		(*Echo OFF*)
		sEchoOff:='ATE0';
		sEchoOff:=CONCAT(sEchoOff,'X');	(*The "X" is a placeholder in the send-string
										for the "CR" (Hex 0D) in the send-Array*)
		MEMCPY(ADR(arEchoOff),ADR(sEchoOff),LEN(sEchoOff)); (*Copy String to ARRAY*)
		arEchoOff[LEN(sEchoOff)]:=16#0D;(*Place the "CR" in the array*)

		(*Mode Text*)
		sLogin:='AT+CMGF=';
		sLogin:=CONCAT(sLogin,'1');
		sLogin:=CONCAT(sLogin,'X');	(*The "X" is a placeholder in the send-string
										for the "CR" (Hex 0D) in the send-Array*)
		MEMCPY(ADR(arLogin),ADR(sLogin),LEN(sLogin)); (*Copy String to ARRAY*)
		arLogin[LEN(sLogin)]:=16#0D;	(*Place the "CR" in the array*)

		nStep	:= 100;


	100:(*Turn Off the Echo*)
		fbSendData(
		pSendData:=ADR(arEchoOff),
		Length:= LEN(sEchoOff),
		TXbuffer:= stTxBuffer);

		IF NOT fbSendData.Busy THEN
			nStep:=110;
		END_IF

		IF  fbSendData.Error<>0 THEN
			bError:= TRUE;
			nErrorID:= fbSendData.Error;
			nStep:=1000;
		END_IF


	110:(*Wait explicitly (by Prefix) for an "OK"-Answer,
		because the echo may still be on or is already switched off, so the answer may differ in length.
		Only ok is possible, any other answer caused by Comm-Error will end in global timeout*)

		fbReceiveData(
		pPrefix:= ADR(arAnswerOK),
		LenPrefix:= 2,
		pReceiveData:= ADR(arEchoOffAnswerRcv),
		SizeReceiveData:= SIZEOF(arEchoOffAnswerRcv),
		Timeout:= t#500ms,
		RXbuffer:= stRxBuffer);

		(*Telegram is received*)
		IF 			fbReceiveData.DataReceived
			AND NOT fbReceiveData.busy
			AND		(arEchoOffAnswerRcv[1]=arAnswerOK[1])
			AND 	(arEchoOffAnswerRcv[2]=arAnswerOK[2])	THEN
						nStep:=200;
		END_IF


	200:(*Send AT+CMGF Command*)
		fbSendData(
		pSendData:=ADR(arLogin),
		Length:= LEN(sLogin),
		TXbuffer:= stTxBuffer);

		IF NOT fbSendData.Busy THEN
			nStep:=210;
		END_IF

		IF  fbSendData.Error<>0 THEN
			bError:= TRUE;
			nErrorID:= fbSendData.Error;
			nStep:=1000;
		END_IF


	210:(*Wait for OK or Err-Answer. Any other answer caused by Comm-Error will end in global timeout*)
		(*Do NOT remove the "0" prefix, because the FB is used previously*)
		fbReceiveData(
		pPrefix:= 0,
		LenPrefix:= 0,
		pReceiveData:= ADR(arLoginAnswerRcv),
		SizeReceiveData:= SIZEOF(arLoginAnswerRcv),
		Timeout:= t#500ms,
		RXbuffer:= stRxBuffer);

		(*Telegram is received*)
		IF 	(fbReceiveData.DataReceived	AND NOT 	fbReceiveData.busy)	THEN
				nStep:=220;
		END_IF


	220:(*Analyze answer*)
		IF		(arLoginAnswerRcv[3]=arAnswerOK[1]) AND (arLoginAnswerRcv[4]=arAnswerOK[2])	THEN
					nStep:=1000;		(*Login successful*)
		ELSIF	(arLoginAnswerRcv[3]=arAnswerErr[1]) AND (arLoginAnswerRcv[4]=arAnswerErr[2])	THEN
					bError:= TRUE;
					nErrorID:= 16#8004;	(*Login failed due to wrong PIN or no Card or already logged in*)
					nStep:=1000;
		ELSE
					bError:= TRUE;
					nErrorID:= 16#8005;	(*Undefined answer*)
					nStep:=1000;
		END_IF


	900:(*Timeout*)
		bError:= TRUE;
		nErrorID:= 16#8001;
		nStep:=1000;


	1000:(*Reset Receive-FB*)
		fbReceiveData(	Reset:=TRUE,RXbuffer:= stRxBuffer);
		tonWaitTime(IN:=TRUE, PT:=t#1000ms);
		IF	tonWaitTime.Q	THEN
			tonWaitTime(IN:=FALSE);
			fbReceiveData(	Reset:=FALSE,RXbuffer:= stRxBuffer);
			nStep:=1010;
		END_IF


	1010:(*Send/Receive successful -> Reset FBs*)
		fbClearComBuffer(buffer:=stRxBuffer);
		fbClearComBuffer(buffer:=stTxBuffer);
		tonWaitTime(IN:=TRUE, PT:=t#1000ms);
		IF	tonWaitTime.Q	THEN
			tonWaitTime(IN:=FALSE);
			nStep:=0;
			bBusy:=FALSE;
		END_IF

	END_CASE;

END_FUNCTION_BLOCK

// ---- 00_FunctionsBlocks/Common/DataProcessing/FB_XorWord.TcPOU
FUNCTION_BLOCK FB_XorWord
// Takes in a Word and its past value and input the bits that have changed and the bits active in 2 arrays of array of bool
VAR_INPUT
	MyNewWord	:WORD;      //Mon nouveau AlarmCode actualisée a chaque temps de Cycle
	MyWord		:WORD;		// AlarmCode du cycle précedent
END_VAR
VAR_OUTPUT
	XORarray 	:ARRAY [0..15] OF BOOL;  //Tableau avec les bits qui ont subit une modif entre MyNewWord et MyWord
	Boolarray	:ARRAY [0..15] OF BOOL; // MyNewWord convertis en Array of BOOL
END_VAR
VAR
	MyXorWord:WORD;
	FB_Word_TO_Bool : FB_WordToArrayOfBool;
END_VAR

// Operateur XOR pour trouver les Bits modifiés
MyXorWord:= Myword XOR MyNewWord;

FB_Word_TO_Bool(MyWord:=MyXorWord,ArrayOfBool=>XORarray);
FB_Word_TO_Bool(MyWord:=MyNewWord,ArrayOfBool=>Boolarray);

END_FUNCTION_BLOCK

// ---- 00_FunctionsBlocks/Common/BoolManagement/FB_WordToArrayOfBool.TcPOU
FUNCTION_BLOCK FB_WordToArrayOfBool
// Transforms a Word in an array of BOOL;
VAR_INPUT
	MyWord	:WORD;
END_VAR
VAR_OUTPUT
	ArrayOfBool: ARRAY [0..15] OF BOOL;
END_VAR

ArrayOfBool[0] := BIT_TO_BOOL(MyWord.0);
ArrayOfBool[1] := BIT_TO_BOOL(MyWord.1);
ArrayOfBool[2] := BIT_TO_BOOL(MyWord.2);
ArrayOfBool[3] := BIT_TO_BOOL(MyWord.3);
ArrayOfBool[4] := BIT_TO_BOOL(MyWord.4);
ArrayOfBool[5] := BIT_TO_BOOL(MyWord.5);
ArrayOfBool[6] := BIT_TO_BOOL(MyWord.6);
ArrayOfBool[7] := BIT_TO_BOOL(MyWord.7);
ArrayOfBool[8] := BIT_TO_BOOL(MyWord.8);
ArrayOfBool[9] := BIT_TO_BOOL(MyWord.9);
ArrayOfBool[10] := BIT_TO_BOOL(MyWord.10);
ArrayOfBool[11] := BIT_TO_BOOL(MyWord.11);
ArrayOfBool[12] := BIT_TO_BOOL(MyWord.12);
ArrayOfBool[13] := BIT_TO_BOOL(MyWord.13);
ArrayOfBool[14] := BIT_TO_BOOL(MyWord.14);
ArrayOfBool[15] := BIT_TO_BOOL(MyWord.15);

END_FUNCTION_BLOCK

// ---- 00_FunctionsBlocks/Beckhoff/Communication/SMS/FB_Extract_Num_Mes.TcPOU
FUNCTION_BLOCK FB_Extract_Num_Mes
// extract phone number from the received message
VAR_INPUT
    InMessage     : STRING(255);
END_VAR
VAR_OUTPUT
    OutDataEntry  :ST_SMSDataSetEntry_Read;
END_VAR
VAR
    ChaineTmp     : STRING(255);
    Num           : STRING(255);
    Pos           : INT;
    Pos1          : INT;
    Pos2          : INT;
    Pos3          : INT;    
	Offset		: INT ; 
END_VAR

//+CMGR: "REC UNREAD","+33776039883",,"18/04/19,18:25:44+08"$R$NBonjour je m'appelle henry$R$N 50
Pos:=FIND(InMessage,',"');
chaineTmp:=MID(InMessage,LEN(InMessage)-21,POS+2);
Pos1:=FIND(chaineTmp,'",,');
Num:=MID(chaineTmp,Pos1-1,1);
Pos3:= FIND(Num,'+');
OutDataEntry.Num:= SEL(Pos3= 0 ,Num ,CONCAT(STR1:= CstPhoneIndicator_G, STR2:= Num) );
Pos2:=FIND(InMessage,'$R$N');
Offset := FIND(MID(InMessage,LEN(InMessage)-Pos2,Pos2+2),'$R$N') ;


OutDataEntry.Message:=MID(InMessage,Offset-1,Pos2+2);//OutDataEntry.Message:=MID(InMessage,LEN(InMessage)-Pos2-3,LEN(InMessage));	// OutDataEntry.Message:=MID(InMessage,LEN(InMessage)-Pos2-3,Pso2+2);

END_FUNCTION_BLOCK

// ---- 04_Application/MAIN/TEST.TcPOU
PROGRAM TEST
VAR
// create an instance for all FB in base project in order to test if there are errors in the FB ()

	moyenne_test : MOYENNE;
	time_Test : TIME := T#5s;
	bTest : BOOL;
	rValue : REAL;

(*
FB_PM_PM5XXX						: FB_PM_PM5XXX ; 
FB_GRID_PLAN						: FB_GRID_PLAN ; 	
FB_CB_AuxMVCB						:FB_CB_AuxMVCB						;
FB_CB_FeederMVCB            		:FB_CB_FeederMVCB            		 ;
FB_CB_GridMVCB               		:FB_CB_GridMVCB               		;
FB_CB_MainHVCB           			:FB_CB_MainHVCB           			;
FB_CB_MainMVCB           			:FB_CB_MainMVCB           			;
FB_CB_MeasureMVCB        			:FB_CB_MeasureMVCB        			;
FB_CB_MVSwitch           	  		:FB_CB_MVSwitch;             		
FB_CB_Switch	               		:FB_CB_Switch;               		
FB_Fan_Basic                		:FB_Fan_Basic                		 ;
FB_FSS                      		:FB_FSS                      		 ;
FB_GRID_Enedis              		:FB_GRID_Enedis              		 ;
FB_GRID_MADI                		:FB_GRID_MADI                		 ;
FB_HVAC_Standard            		:FB_HVAC_Standard            		          ;
FB_HVAC_MADI                		:FB_HVAC_MADI                		 ;
FB_PM_520x230               		:FB_PM_520x230               		 ;
FB_PM_A40                   		:FB_PM_A40                   		 ;
FB_PM_ION7650               		:FB_PM_ION7650               		 ;
FB_PM_Janitza               		:FB_PM_Janitza               		 ;
FB_PM_PM3250                		:FB_PM_PM3250                		 ;
FB_PM_SM103E                		:FB_PM_SM103E                		 ;
FB_ProtectRelay_DM2     			:FB_ProtectRelay_DM2     		;
FB_ProtectRelay_PACE100ST    		:FB_ProtectRelay_PACE100ST    		;
FB_ProtectRelay_REF615       		:FB_ProtectRelay_REF615       		;
FB_ProtectRelay_SEPAM10a     		:FB_ProtectRelay_SEPAM10a     		;
FB_ProtectRelay_SepamS48     		:FB_ProtectRelay_SepamS48     		;
FB_ProtectRelay_SepamT20     		:FB_ProtectRelay_SepamT20     		;
FB_ProtectRelay_VIP410       		:FB_ProtectRelay_VIP410       		;
FB_ProtectRelay_WIP1         		:FB_ProtectRelay_WIP1         		;
FB_ANA_Irra_Fx               		:FB_ANA_Irra_Fx               		;
FB_ANA_SMP1X                 		:FB_ANA_SMP1X                 		;
FB_ANA_AllInOne              		:FB_ANA_AllInOne              		    ;
FB_TOR_CB                    		:FB_TOR_CB                    		;
FB_TOR_DS                    		:FB_TOR_DS                    		;
FB_TOR_ES                    		:FB_TOR_ES                    		;
FB_TOR_Fuse                  		:FB_TOR_Fuse                  		;
FB_TOR_Rain                			:FB_TOR_Rain                			;
FB_TOR_SD                    		:FB_TOR_SD                    		;
FB_TOR_Spd                   		:FB_TOR_Spd                   		;
FB_TOR_ToS                   		:FB_TOR_ToS                   		;
FB_EM_Pulse                  		:FB_EM_Pulse                  		      ;
FB_Transfo_HVCom             		:FB_Transfo_HVCom             		;
FB_Transfo_MV                		:FB_Transfo_MV                		;
FB_Transfo_MVCom             		:FB_Transfo_MVCom             		;
FB_UPS_CXC                   		:FB_UPS_CXC                   		;
FB_UPS_ENERIS                		:FB_UPS_ENERIS                		;
FB_BAT_KP_MK1						: FB_BAT_KP_MK1					; 
//FB_BAT_M3							: FB_BAT_M3       					;          
FB_BAT_Saft                 		: FB_BAT_Saft                      ;
FB_BAT_Sams                 		: FB_BAT_Sams                      ;

FB_Datalogger_SchSkid       		: FB_Datalogger_SchSkid            ;

FB_HVAC_MeAcMbs1            		: FB_HVAC_MeAcMbs1                 ;
*)
FB_INV_Huawei_SL            		: FB_INV_Huawei_SL                 ;

FB_INV_Huawei_Sun2000KtlMo  		: FB_INV_Huawei_Sun2000KtlMo       ;
FB_INV_JemaIFX6             		: FB_INV_JemaIFX6                  ;
FB_INV_Power_One            		: FB_INV_Power_One                 ;
FB_INV_Sch4400              		: FB_INV_Sch4400                   ;
FB_INV_SmaSCXXXXCP_HE       		: FB_INV_SmaSCXXXXCP_HE            ;
FB_INV_SmaSCXXXXUP_US       		: FB_INV_SmaSCXXXXUP_US            ;
(*
FB_IPC                      		: FB_IPC                           ;
FB_PM_Digiware              		: FB_PM_Digiware                   ;
FB_PM_PM800                 		: FB_PM_PM800                      ;
FB_PM_Prometer              		: FB_PM_Prometer                   ;
FB_PM_Q100                  		: FB_PM_Q100                       ;
FB_PCS_Jema_IBX3            		: FB_PCS_Jema_IBX3                 ;
FB_PCS_PE                   		: FB_PCS_PE                        ;
FB_PCS_Sma_SCS3450UP        		: FB_PCS_Sma_SCS3450UP             ;
FB_PPC_SmaKita              		: FB_PPC_SmaKita                   ;
FB_ProtectRelay_Siprotec    	    : FB_ProtectRelay_Siprotec         ;
FB_ProtectRelay_Flair23DM   	    : FB_ProtectRelay_Flair23DM        ;
FB_ProtectRelay_MaxI        	    : FB_ProtectRelay_MaxI             ;
FB_ProtectRelay_NSXCB       	    : FB_ProtectRelay_NSXCB            ;
FB_Router                   	    : FB_Router                        ;
FB_ANA_IO                   	    : FB_ANA_IO                        ;
FB_ANA_DustIQ               	    : FB_ANA_DustIQ                    ;

FB_TOR_Digicode             	    : FB_TOR_Digicode                  ;
FB_TOR_Standard             	    : FB_TOR_Standard                  ;
FB_TOR_MS                   	    : FB_TOR_MS                        ;
FB_TOR_VP                   	    : FB_TOR_VP                        ;
FB_TAC                      	    : FB_TAC                           ;
FB_NCU_Axial                	    : FB_NCU_Axial                     ;
FB_UPS_PS10048              	    : FB_UPS_PS10048                   ;
FB_PM_ION9200						: FB_PM_ION9200 ; 	
	

FB_PPC_PE							: FB_PPC_PE ; 
FB_UPS_MCSU4 						: FB_UPS_MCSU4 ; 
FB_ProtectRelay_SMNS7SL86 			: FB_ProtectRelay_SMNS7SL86 ; 
*)
FB_INV_PE_HEMK : FB_INV_PE_HEMK ; 
	FB_INV_PE_HEMG3 : FB_INV_PE_HEMG3 ; 
END_VAR


moyenne_test(
	In_fenetre_mesure := time_Test,
	In_synchro := CalLocalTimeStruct.wSecond MOD 5 = 0,
	In_valeur := word_to_real(CalLocalTimeStruct.wSecond)
);
moyenne_test.Calcul();

(*
FB_GRID_PLAN.M_Execute() ; 
FB_CB_AuxMVCB.M_Execute() ; 					
FB_CB_FeederMVCB.M_Execute() ; 			            	
FB_CB_GridMVCB.M_Execute() ; 			               	
FB_CB_MainHVCB.M_Execute() ; 			           		
FB_CB_MainMVCB.M_Execute() ; 			           		
FB_CB_MeasureMVCB.M_Execute() ; 			        		
FB_CB_MVSwitch.M_Execute() ; 			             	
FB_CB_Switch.M_Execute() ; 			               	
FB_Fan_Basic.M_Execute() ; 		                	
FB_FSS.M_Execute() ; 		                      	
FB_GRID_Enedis.M_Execute() ; 		              	
FB_GRID_MADI.M_Execute() ; 		                	
FB_HVAC_Standard.M_Execute() ; 		            	
FB_HVAC_MADI.M_Execute() ; 		                	
FB_PM_520x230.M_Execute() ; 		               	
FB_PM_A40.M_Execute() ; 		                   	
FB_PM_ION7650.M_Execute() ; 		               	
FB_PM_Janitza.M_Execute() ; 		               	
FB_PM_PM3250.M_Execute() ; 		                	
FB_PM_SM103E.M_Execute() ; 		                	
FB_ProtectRelay_DM2.M_Execute() ; 		     		
FB_ProtectRelay_PACE100ST.M_Execute() ; 		    	
FB_ProtectRelay_REF615.M_Execute() ; 		       	
FB_ProtectRelay_SEPAM10a.M_Execute() ; 		     	
FB_ProtectRelay_SepamS48.M_Execute() ; 		     	
FB_ProtectRelay_SepamT20.M_Execute() ; 		     	
FB_ProtectRelay_VIP410.M_Execute() ; 		       	
FB_ProtectRelay_WIP1.M_Execute() ; 		         	
FB_ANA_Irra_Fx.M_Execute() ; 		               	
FB_ANA_SMP1X.M_Execute() ; 		                 	
FB_ANA_AllInOne.M_Execute() ; 		              	
FB_TOR_CB.M_Execute() ; 		                    	
FB_TOR_DS.M_Execute() ; 		                    	
FB_TOR_ES.M_Execute() ; 		                    	
FB_TOR_Fuse.M_Execute() ; 		                  	
FB_TOR_Rain.M_Execute() ; 		                		
FB_TOR_SD.M_Execute() ; 		                    	
FB_TOR_Spd.M_Execute() ; 		                   	
FB_TOR_ToS.M_Execute() ; 		                   	
FB_EM_Pulse.M_Execute() ; 		                  	
FB_Transfo_HVCom.M_Execute() ; 		             	
FB_Transfo_MV.M_Execute() ; 		                	
FB_Transfo_MVCom.M_Execute() ; 		             	
FB_UPS_CXC.M_Execute() ; 		                   	
FB_UPS_ENERIS.M_Execute() ; 		                	
FB_BAT_KP_MK1.M_Execute() ; 							
FB_BAT_M3.M_Execute() ; 								
FB_BAT_Saft.M_Execute() ; 		                 	
FB_BAT_Sams.M_Execute() ; 		                 	
FB_Datalogger_IOWIT.M_Execute() ; 		         	
FB_Datalogger_PPCVerrerie.M_Execute() ; 		   	
FB_Datalogger_SchSkid.M_Execute() ; 		       	
FB_Datalogger_SENECA.M_Execute() ; 		        	
FB_HVAC_MeAcMbs1.M_Execute() ; 		            	
*)
FB_INV_Huawei_SL.M_Execute() ; 		            	
FB_INV_Huawei_Sun2000KtlMo.M_Execute() ; 		  	
FB_INV_JemaIFX6.M_Execute() ; 		             	
FB_INV_Power_One.M_Execute() ; 		            	
FB_INV_Sch4400.M_Execute() ; 		              	
FB_INV_SmaSCXXXXCP_HE.M_Execute() ; 		       	
FB_INV_SmaSCXXXXUP_US.M_Execute() ; 		       	


(*
FB_IPC.M_Execute() ; 		                      	
FB_PM_Digiware.M_Execute() ; 		              	
FB_PM_PM800.M_Execute() ; 		                 	
FB_PM_Prometer.M_Execute() ; 		              	
FB_PM_Q100.M_Execute() ; 		                  	
FB_PCS_Jema.M_Execute() ; 		                 	
FB_PCS_Jema_IBX3.M_Execute() ; 		            	
FB_PCS_PE.M_Execute() ; 		                   	
FB_PCS_Sma_SCS3450UP.M_Execute() ; 		       	
FB_PPC_SmaKita.M_Execute() ; 		              	
FB_ProtectRelay_Siprotec.M_Execute() ; 		    	
FB_ProtectRelay_Flair23DM.M_Execute() ; 		   	
FB_ProtectRelay_MaxI.M_Execute() ; 		        	
FB_ProtectRelay_NSXCB.M_Execute() ; 		       	
FB_Router.M_Execute() ; 		                   	
FB_ANA_IO.M_Execute() ; 		                   	
FB_ANA_Irra_Fx.M_Execute() ; 		              	
FB_ANA_DustIQ.M_Execute() ; 		               	
FB_ANA_SMP1X.M_Execute() ; 		               	
FB_TOR_Digicode.M_Execute() ; 		             	
FB_TOR_Standard.M_Execute() ; 		             	
FB_TOR_MS.M_Execute() ; 		                   	
FB_TOR_VP.M_Execute() ; 		                   	
FB_TAC.M_Execute() ; 		                      	
FB_EM_Pulse.M_Execute() ; 		                 	
FB_NCU_Axial.M_Execute() ; 		                	
FB_UPS_PS10048.M_Execute() ; 		              	
FB_PM_PM5XXX.M_Execute() ; 
FB_PM_ION9200.M_Execute() ; 
FB_PPC_PE.M_Execute() ; 

				  				
FB_UPS_MCSU4.M_Execute() ;  				
FB_ProtectRelay_SMNS7SL86.M_Execute() ;  	
*)
FB_INV_PE_HEMG3.M_Execute() ;  
FB_INV_PE_HEMK.M_Execute();

END_PROGRAM

// ---- 00_FunctionsBlocks/Beckhoff/DataProcessing/MOYENNE.TcPOU
FUNCTION_BLOCK MOYENNE
VAR_INPUT
	In_valeur: REAL;
	In_synchro: BOOL;
	In_fenetre_mesure: TIME;
END_VAR
VAR_OUTPUT
	Out_fenetre_mesure: TIME;
	Out_fin: BOOL;
	Out_Moyenne_0: REAL;
	Out_Moyenne_1: REAL;
END_VAR
VAR
	F_Fenetre_mesure_active: F_TRIG;
	R_In_Synchro: R_TRIG;
	TOF_0: TOF;
	Fenetre_mesure_active: BOOL;
	Nbr_valeur_mesure: REAL;
END_VAR

ACTION Calcul:
(* Gestion des fronts montants et front descendants *)

	R_In_Synchro(CLK := In_Synchro);
	F_Fenetre_mesure_active(CLK := Fenetre_mesure_active);

(* Traitements *)

	IF R_In_Synchro.Q THEN  (* Initialisation des valeurs au lancement de la synchronisation *)
	
		Out_fin:=False; 
		Nbr_valeur_mesure:=0.0; (* RAZ nbr de cycle automate *)
	
	END_IF;
	

	TOF_0 (IN := R_In_Synchro.Q,(* Gestion de la fenêtre de mesure  *)
		  PT := In_fenetre_mesure,
		  Q => Fenetre_mesure_active,
		  ET => Out_fenetre_mesure);
	
	IF Fenetre_mesure_active  THEN (* Traitement durant la fenêtre de mesure *) 
		
		Out_Moyenne_0:=(Out_Moyenne_0*Nbr_valeur_mesure+In_valeur)/(Nbr_valeur_mesure+1.0); (* calcul moyenne *)
	
		Nbr_valeur_mesure:=Nbr_valeur_mesure+1.0; (* calcul nbr de cycle automate *)
	
	ELSIF F_Fenetre_mesure_active.Q THEN (* Traitement en fin de fenêtre de mesure *)
	
		Out_fin:=true;
		Out_Moyenne_1:=Out_Moyenne_0; (* Sauvegarde de la moyenne calculée *)
		Out_Moyenne_0:=0.0; (* RAZ moyenne calculée *)
	
	End_if;
END_ACTION

END_FUNCTION_BLOCK

// ---- 01_Equipement_Library/Inverter/FB_INV_Huawei_SL.TcPOU
FUNCTION_BLOCK FB_INV_Huawei_SL EXTENDS FB_INV_Base
//////////////////
// SmartLogger Huawei
//////////////////

VAR_INPUT PERSISTENT
	// Parameters of the Object (instance specific)
	{attribute 'OPC.UA.DA' := '1'}  
	ParamIpAddress		   : STRING 	:= '127.0.0.1'; (* (NA)Config: IP Adress of PV INverter*)
	{attribute 'OPC.UA.DA' := '1'} 
	ParamUnitID 			: BYTE  := 0; 			  	(* (NA)   Modbus Unit ID. *)
	ParamNbINV				: BYTE:=1 ; 				(* Number of inverters behind the smartlogger *)
	{attribute 'OPC.UA.DA' := '1'}              		
	ParamnTcpPort			: UINT := 502;				(* TCP port number *)
	ParamPnomINV			: REAL:=60; 				(* (kW) Nominal Power For one inverter *)
	ParamSLNum				: BYTE ; 					(* (NA) Config :Numerous of the ESS in the PP*)
	ParamID_PTR				: UINT;						(* (NA) ID of the PTR where Smartlogger is located*)
	
	
		MesDataExd	AT %Q*		: INV_Huawei_SL;
	
END_VAR

VAR_OUTPUT
	//Child objects
	
END_VAR

VAR

	// M_READ VARIABLES//


//		FB_ModbusRead_I1          	: ARRAY[1..CstNbINVperPTR_G] OF  FB_ModbusRead ; 		// (NA) FB for Modbus Reading
		FB_ModbusRead_I2          	: FB_ModbusRead ; 										// (NA) FB for Modbus Reading
		FB_ModbusRead_I3          	: FB_ModbusRead ; 										// (NA) FB for Modbus Reading
			
//		MesBlock1_Temp 				: ARRAY[1..CstNbINVperPTR_G] OF ARRAY[0..24]  OF WORD; 	// (NA) Temporary Block with multiple modbus reading (Caution : Double Word variables)
//		MesBlock1_Temp 				: ARRAY[0..25*CstNbINVperPTR_G-1]  OF WORD; 			// (NA) Temporary Block with multiple modbus reading (Caution : Double Word variables)
		MesBlock2_Temp 				: ARRAY[0..56] OF WORD;									// (NA) Temporary Block with multiple modbus reading (Caution : Double Word variables)
		MesBlock3_Temp 				: ARRAY[0..14] OF WORD;									// (NA) Temporary Block with multiple modbus reading (Caution : Double Word variables)
                                                                                    		
		                                                                            		
//		MesModbusReadAlarm 		  	: ARRAY[1..CstNbINVperPTR_G] OF BOOL ; 					// (NA) Modbus Read Alarm for all modbus frames		
		MesModbusReadAlarm2 		: BOOL ; 												// (NA) Modbus Read Alarm for all modbus frames			
		MesModbusReadAlarm3 		: BOOL ; 												// (NA) Modbus Read Alarm for all modbus frames			

//		MesModbusAlarmCode			: ARRAY[1..CstNbINVperPTR_G] OF UDINT;					// (NA) Modbus Read Alarm Code
		MesModbusAlarmCode2			: UDINT;												// (NA) Modbus Read Alarm Code
		MesModbusAlarmCode3			: UDINT;												// (NA) Modbus Read Alarm Code

	
	// M_CURTAIL VARIABLES //
		FB_ModbusWrite_I2 		  	: FB_ModbusWrite ; 										// (NA) Functionnal Block for Writing Curtail limit through modbus
		FB_ModbusWrite_I3 		  	: FB_ModbusWrite ; 										// (NA) Functionnal Block for Writing Curtail limit through modbus	
		MesModbusWriteCode          : UDINT ; 												// (NA) Modbus Write Alarm Code 			 
		MesModbusWriteCode2         : UDINT ; 												// (NA) Modbus Write Alarm Code 
	                                                                           		
		MesModbusCurtailAlarm		: BOOL ;				   								// (NA) Modbus Write Curtail Alarm 
		MesModbusCurtailAlarm2		: BOOL ;				   								// (NA) Modbus Write Curtail Alarm 
		WriteBlock_Temp 	AT %Q*	: ARRAY[0..3] OF WORD;				 					// Temporary Block with multiple modbus writing	 
		
END_VAR

METHOD M_AlarmManagement
//////////////////
// Manages IntelliGen Alarms
/////////////////

VAR 
	// Method local variables (reinitialized at each cycle) 
	FB_AlarmCodeManager : FB_AlarmCodeManager ; 

	KK					: BYTE;		// For Loop 
	
	ComWarning			: BOOL;		// Aggregated Wcommunication warning
	ComAlarm			: BOOL;		// Aggregated communication Alarm
	ComINVWarning			: BOOL;		// Aggregated Wcommunication warning
	ComINVAlarm			: BOOL;		// Aggregated communication Alarm
	
	INVAlarm			: BOOL ; // At least one inverter has an alarm
END_VAR
//COMMUNICATION//
	CalModbusWriteAlarm := MesModbusCurtailAlarm ; 
	
	ComWarning 			:= MesModbusCurtailAlarm ;			// At least one modbus trame did not work
	ComAlarm			:= TRUE;						// All modbus trame did not work
	
		ComWarning 	:= ComWarning OR  MesModbusReadAlarm2 OR MesModbusReadAlarm3; // Smart logger LOC
		ComAlarm	:= ComAlarm  AND MesModbusReadAlarm2 AND MesModbusReadAlarm3; 
		
//		ComINVWarning := FALSE ; // LOC with inverters
//		ComINVAlarm	 := TRUE ; 
//		INVAlarm		:=FALSE ; 
		
(*	FOR KK:=1 TO ParamNbINV DO 
		ComINVWarning 	:= ComINVWarning OR MesDataExd.MesData.LExd.MesDataExd.MesData.NV[KK].CalComAlarm;
	    ComINVAlarm	:= ComINVAlarm  AND MesDataExd.MesData.LExd.MesDataExd.MesData.NV[KK].CalComAlarm ;
		INVAlarm := INVAlarm AND MesDataExd.MesData.LExd.MesDataExd.MesData.NV[KK].MesAlarm ;
	END_FOR
	*)	
	//Warning
	MesWarningCom 	:= ComWarning ;  
	//Alarm
	TON_ComAlarm(IN:= ComAlarm , PT:= ParamTempoComAlarm, Q=> MesDataExd.MesData.MesAlarmCom) ;	

// ALARM CODE //

// Attention une alarm doit être mise en commentaire de la manière suivante (* *), l'utilisation du // pose pb sur Bazefield 

	FB_AlarmCodeManager(
		bAlarm1			:= MesDataExd.MesData.MesState_Inv=6 ,	// Smart Logger general alarm (desactivate if LOC)  
		bAlarm2			:= MesDataExd.MesData.MesAlarmCom,  // Loss of communication with smart logger #COM
		bAlarm3			:=ComINVAlarm AND NOT MesWarningCom , 		// LOC with all inverters while they were connected
		bAlarm4			:=MesModbusCurtailAlarm, 		// 
		bAlarm5			:=FALSE, 
		bAlarm6			:=FALSE, 
		bAlarm7			:=FALSE, 
		bAlarm8			:=FALSE, 
		bAlarm9			:=FALSE, 
		bAlarm10		:=FALSE, 
		bAlarm11		:=FALSE, 
		bAlarm12		:=FALSE, 
		bAlarm13		:=FALSE, 
		bAlarm14		:=FALSE, 													// 
		bAlarm15		:= FALSE , 									// Command Alarm in case of intervention
		wAlarmCode		=>MesDataExd.MesData.MesAlarmCode);

// WARNING CODE //
	FB_AlarmCodeManager(
 		bAlarm1			:= ComINVWarning,								// At least one inverter has a loss of communication
		bAlarm2			:= CalCompareWarningCurtail,					// Measured Power above curtail Power 
		bAlarm3			:= MesWarningCom,								// Bad communication #COM
		bAlarm4			:=INVAlarm, 		// At least one inverter has an alarm
		bAlarm5			:=FALSE, 
		bAlarm6			:=FALSE, 
		bAlarm7			:=FALSE, 
		bAlarm8			:=FALSE, 
		bAlarm9			:=FALSE, 
		bAlarm10		:=FALSE, 
		bAlarm11		:=FALSE, 
		bAlarm12		:=FALSE, 
		bAlarm13		:=FALSE, 
		bAlarm14		:=FALSE, 
		bAlarm15		:=FALSE, 
		wAlarmCode		=>MesDataExd.MesData.MesWarningCode);	

// EVENT CODE //
	FB_AlarmCodeManager(
		bAlarm1			:= RS_StartStop.Q1, 			// Start command
		bAlarm2			:= NOT RS_StartStop.Q1, 		// Stop command
		bAlarm3			:= MesDataExd.MesData.MesState_Inv=2 OR MesDataExd.MesData.MesState_Inv=3, 		// Curtailing is ON
		bAlarm4			:= FALSE, 		// 
		bAlarm5			:= FALSE, 
		bAlarm6			:= FALSE, 
		bAlarm7			:= FALSE, 
		bAlarm8			:= FALSE, 
		bAlarm9			:= FALSE, 
		bAlarm10		:= FALSE, 
		bAlarm11		:= FALSE, 
		bAlarm12		:= FALSE, 
		bAlarm13		:= FALSE, 
		bAlarm14		:= FALSE, 
		bAlarm15		:= FALSE, 
		wAlarmCode		=>MesDataExd.MesData.MesEventCode);
END_METHOD

METHOD M_CP
//////////////////
//  Emulator
/////////////////

VAR 
	// Method local variables (reinitialized at each cycle) 
	
END_VAR


SUPER^.M_CP() ; 




Trig_Cmd_Read(CLK:=IN_CmdToggleRead);
Trig_Cmd_Write(CLK:=IN_CmdToggleWrite);
	
IF Trig_Cmd_Read.Q THEN
	IN_CmdToggleRead := FALSE;
	MesDataExd.MesData.MesCP_Read := NOT MesDataExd.MesData.MesCP_Read;
END_IF


IF Trig_Cmd_Write.Q THEN
	IN_CmdToggleWrite := FALSE;
	MesDataExd.MesData.MesCP_Write := NOT MesDataExd.MesData.MesCP_Write;
END_IF
END_METHOD

{attribute 'object_name' := 'M_Curtail'}
METHOD M_Curtail
//////////////////
// Write Curtail Command through modbus to PV inverters.  
//////////////////
VAR 
	// Method local variables (reinitialized at each cycle) 
	
	Threshold 			 : INT:=5 ;					// (0-100) Change percentage of Range to trigger the write commAND  

	CHECK				 : BOOL; 					// Check if changes. 
	WriteCmd 			 : BOOL;					// Modbus Write Rising Edge 
	
	SetptPlimit_Temp: ARRAY[0..1] OF WORD;
	SetptQlimit_Temp: ARRAY[0..1] OF WORD;
	
	WriteBlock_Temp1 				: ARRAY[0..1] OF WORD; 	// Temporary Block with multiple modbus writing	 
	WriteBlock_Temp2 				: ARRAY[0..1] OF WORD; 	// Temporary Block with multiple modbus writing	
	
	Split		: FB_SplitRealToWords ; 
	
	CHECK2: BOOL;

	CalInhibeWrite: BOOL;


	Quantity: BYTE;
END_VAR
// MODBUS VARIABLE FORMATING //
MesDataExd.MesData.OUT_SetptPLimit	:= MIN(MesDataExd.MesSetptPMax,MAX(0, IN_SetptPlimit)) ; 
MesDataExd.MesData.OUT_SetptQ	:= MIN(MesDataExd.MesSetptQMax , MAX(MesDataExd.MesSetptQMin , IN_SetptQ)) ; 
		
	
	Split(IN:= MesDataExd.MesData.OUT_SetptPLimit*10.0 , OUT=>SetptPlimit_Temp ) ;   //Between 0 and 100% Pmax
	Split(IN:= MesDataExd.MesData.OUT_SetptQ*10.0 , OUT=>SetptQlimit_Temp ) ; // Cosphi limité à 0.8
	
	
	WriteBlock_Temp1[0] := SetptPlimit_Temp[0] ; 
	WriteBlock_Temp1[1] := SetptPlimit_Temp[1] ; 
	WriteBlock_Temp2[0] := SetptQlimit_Temp[0] ; 
	WriteBlock_Temp2[1] := SetptQlimit_Temp[1] ; 

// MODBUS REQUEST //	
	// Modbus Blocks write
	FB_ModbusWrite_I2(
		pSrcAddr 			:= ADR(WriteBlock_Temp1) ,
		cbLength			:= SIZEOF(WriteBlock_Temp1) , 
		nQuantity 			:= 2,
		Reset				:= CmdClearFault_G, 
		sIPAddr				:=ParamIpAddress ,
		nTCPport			:= ParamnTcpPort ,  
		nUnitID				:=ParamUnitID , 
		nMBAddr				:=40424 , 
		tTimeout			:=ParamTimeout ,
		WriteCmd			:=ClockWrite AND MesDataExd.MesData.MesCP_Write, 
		ModbusWriteAlarm	=>MesModbusCurtailAlarm , 
		ErrorId				=> MesModbusWriteCode); 

	FB_ModbusWrite_I3(
		pSrcAddr 			:= ADR(WriteBlock_Temp2) ,
		cbLength			:= SIZEOF(WriteBlock_Temp2) , 
		nQuantity 			:= 2,
		Reset				:= CmdClearFault_G, 
		sIPAddr				:=ParamIpAddress ,
		nTCPport			:= ParamnTcpPort ,  
		nUnitID				:=ParamUnitID , 
		nMBAddr				:=40426 , 
		tTimeout			:=ParamTimeout ,
		WriteCmd			:=ClockWrite AND MesDataExd.MesData.MesCP_Write, 
		ModbusWriteAlarm	=>MesModbusCurtailAlarm2 , 
		ErrorId				=> MesModbusWriteCode2); 

	IF FB_ModbusWrite_I2.Completed THEN
		MesDataExd.OUT_SetptPlimit 	:= IN_SetptPlimit ;
		MesDataExd.OUT_SetptQlimit	:= IN_SetptQ;
	END_IF
END_METHOD

METHOD M_Init
VAR_INPUT
END_VAR

VAR

END_VAR
 MesDataExd.OUT_SetptPlimit := 9999999 ; // initialize to absurd value , to force a write of setpoint at startup . 
MesDataExd.OUT_SetptQlimit	:= 9999999 ; // initiali
END_METHOD

{attribute 'object_name' := 'M_Read'}
METHOD M_Read
//////////
// Read Method for SMA : Modbus reading
//////////
VAR
	// Method local variables (reinitialized at each cycle) 
	MW 					: FB_MergeWordsToDint; 
	KK					: BYTE;						 // Index to loop over modbus blocks. 	

END_VAR
// Version table de com : Issu 37

IF	MesDataExd.MesData.MesCP_Read THEN	
	
	// Datalogger //
		//INITIALIZING MODBUS REQUESTS //
		FB_ModbusRead_I2(ClockRead:= ClockRead AND MesDataExd.MesData.MesCP_Read, Reset:= CmdClearFault_G ,sIPAddr:=ParamIpAddress , nUnitID:= ParamUnitID, tTimeout:= ParamTimeout,nTcpPort := ParamnTcpPort);
		FB_ModbusRead_I3(ClockRead:= ClockRead AND MesDataExd.MesData.MesCP_Read, Reset:= CmdClearFault_G ,sIPAddr:=ParamIpAddress , nUnitID:= ParamUnitID, tTimeout:= ParamTimeout,nTcpPort := ParamnTcpPort);
	
	// MODBUS REQUEST//
		FB_ModbusRead_I2(
			nQuantity		:= 57, 
			nMBAddr			:= 40521, 
			cbLength		:= SIZEOF(MesBlock2_Temp) , 
			pDestAddr		:= ADR(MesBlock2_Temp) , 
			ModbusReadAlarm	=>MesModbusReadAlarm2 , 
			ErrorId			=> MesModbusAlarmCode2);
			
		FB_ModbusRead_I3(
			nQuantity		:= 15, 
			nMBAddr			:= 40685, 
			cbLength		:= SIZEOF(MesBlock3_Temp) , 
			pDestAddr		:= ADR(MesBlock3_Temp) , 
			ModbusReadAlarm	=>MesModbusReadAlarm3 , 
			ErrorId			=> MesModbusAlarmCode3);		
			
	
	// MODBUS BLOCKS SEPARATION	
			MW(WORD_STRONG:= MesBlock2_Temp[0], WORD_WEAK := MesBlock2_Temp[1],SIGNED:=FALSE, FIX:=3 , SIZE:=2, VAR_OUT := MesDataExd.MesData.MesPdc);
	
			MW(WORD_STRONG:= MesBlock2_Temp[4], WORD_WEAK := MesBlock2_Temp[5],SIGNED:=TRUE, FIX:=3 , SIZE:=2, VAR_OUT := MesDataExd.MesData.MesP);
			MW(WORD_STRONG:= MesBlock2_Temp[11],SIGNED:=TRUE, FIX:=3 , SIZE:=1, VAR_OUT := MesDataExd.MesData.MesCosPhi);
	
			MW(WORD_STRONG:= MesBlock2_Temp[23], WORD_WEAK := MesBlock2_Temp[24],SIGNED:=TRUE, FIX:=3 , SIZE:=2, VAR_OUT := MesDataExd.MesData.MesQ);
			MW(WORD_STRONG:= MesBlock2_Temp[33], WORD_WEAK := MesBlock2_Temp[34],SIGNED:=TRUE, FIX:=1 , SIZE:=2, VAR_OUT := MesDataExd.MesData.MesIdc);
			MW(WORD_STRONG:= MesBlock2_Temp[39], WORD_WEAK := MesBlock2_Temp[40],SIGNED:=FALSE, FIX:=1 , SIZE:=2, VAR_OUT := MesDataExd.MesETot);
			MW(WORD_STRONG:= MesBlock2_Temp[41], WORD_WEAK := MesBlock2_Temp[42],SIGNED:=FALSE, FIX:=1 , SIZE:=2, VAR_OUT := MesDataExd.MesEDay);
		MesDataExd.MesData.MesState_Inv:= MesBlock2_Temp[45];
			
			MW(WORD_STRONG:= MesBlock2_Temp[51],SIGNED:=TRUE, FIX:=0 , SIZE:=1, VAR_OUT := MesDataExd.MesI1);
			MW(WORD_STRONG:= MesBlock2_Temp[52],SIGNED:=TRUE, FIX:=0 , SIZE:=1, VAR_OUT := MesDataExd.MesI2);
			MW(WORD_STRONG:= MesBlock2_Temp[53],SIGNED:=TRUE, FIX:=0 , SIZE:=1, VAR_OUT := MesDataExd.MesI3);
			MW(WORD_STRONG:= MesBlock2_Temp[54],SIGNED:=FALSE, FIX:=1 , SIZE:=1, VAR_OUT := MesDataExd.MesU12);
			MW(WORD_STRONG:= MesBlock2_Temp[55],SIGNED:=FALSE, FIX:=1 , SIZE:=1, VAR_OUT := MesDataExd.MesU23);
			MW(WORD_STRONG:= MesBlock2_Temp[56],SIGNED:=FALSE, FIX:=1 , SIZE:=1, VAR_OUT := MesDataExd.MesU31);
		
		MW(WORD_STRONG:= MesBlock2_Temp[51],SIGNED:=TRUE, FIX:=0 , SIZE:=1, VAR_OUT := MesDataExd.MesI1);
		MW(WORD_STRONG:= MesBlock2_Temp[52],SIGNED:=TRUE, FIX:=0 , SIZE:=1, VAR_OUT := MesDataExd.MesI2);
		MW(WORD_STRONG:= MesBlock2_Temp[53],SIGNED:=TRUE, FIX:=0 , SIZE:=1, VAR_OUT := MesDataExd.MesI3);
		MW(WORD_STRONG:= MesBlock2_Temp[54],SIGNED:=FALSE, FIX:=1 , SIZE:=1, VAR_OUT := MesDataExd.MesU12);
		MW(WORD_STRONG:= MesBlock2_Temp[55],SIGNED:=FALSE, FIX:=1 , SIZE:=1, VAR_OUT := MesDataExd.MesU23);
		MW(WORD_STRONG:= MesBlock2_Temp[56],SIGNED:=FALSE, FIX:=1 , SIZE:=1, VAR_OUT := MesDataExd.MesU31);
		
		
		
	
		// Block 3
		MW(WORD_STRONG:= MesBlock3_Temp[0], SIGNED:=FALSE, FIX:=2 , SIZE:=1, VAR_OUT := MesDataExd.MesEff);
		MW(WORD_STRONG:= MesBlock3_Temp[8],WORD_WEAK := MesBlock3_Temp[9], SIGNED:=FALSE, FIX:=2 , SIZE:=2, VAR_OUT := MesDataExd.MesSetptQMax);
		MW(WORD_STRONG:= MesBlock3_Temp[10],WORD_WEAK := MesBlock3_Temp[11], SIGNED:=TRUE, FIX:=2 , SIZE:=2, VAR_OUT := MesDataExd.MesSetptQMin);
		MW(WORD_STRONG:= MesBlock3_Temp[12],WORD_WEAK := MesBlock3_Temp[13], SIGNED:=FALSE, FIX:=2 , SIZE:=2, VAR_OUT := MesDataExd.MesSetptPMax);
	MesDataExd.MesOn	:= 	MesBlock3_Temp[14].0 ; 	
	


END_IF
	
// Properties update
	ParamPn := ParamPnomINV * ParamNbINV ;
END_METHOD

METHOD M_StartStop
//////////////////
// Start and Stop AMG
/////////////////
VAR 
	// Method local variables (reinitialized at each cycle) 

END_VAR
END_METHOD

METHOD M_StateManager
//////////////////
// Detect which is the state of the inverter. IF loss of communication MesState =0 , the last inverter state is kept .  
/////////////////

VAR 
	// Method local variables (reinitialized at each cycle) 

	
END_VAR

MesDataExd.MesData.MesState 			:= 0  ; 
//O=Stopped, 1 = MPPT, 2 = Sleeping, 3 = Starting, 4 = Throttled, 5 = Shutting down, 6 = Fault, 7 = Standby


IF MesDataExd.MesData.MesState_Inv = 0 THEN //idle 
	// Standby
	MesDataExd.MesData.MesState .7 		:= 1 ;
ELSIF  MesDataExd.MesData.MesState_Inv = 1 THEN //on grid 

	// ON State
	MesDataExd.MesData.MesState.1 		:= 1 ; 		// At least one inverter is feeding power to the grid .

ELSIF  MesDataExd.MesData.MesState_Inv = 2 OR  MesDataExd.MesData.MesState_Inv = 3  THEN //on grid 
 	MesDataExd.MesData.MesState.4 		:= 1 ; 		// At least one inverter is feeding power to the grid .
	
ELSIF  MesDataExd.MesData.MesState_Inv = 4 OR MesDataExd.MesData.MesState_Inv = 5 THEN // planned outage , power limit outage 
	 MesDataExd.MesData.MesState .0 		:= 1 ;
	 
ELSIF  MesDataExd.MesData.MesState_Inv = 6 THEN //fault outage
	 MesDataExd.MesData.MesState .6 		:= 1 ;
ELSE // Communication interrupt 
	// OFF State  
	MesDataExd.MesData.MesState .1 		:= 1 ; 
	
END_IF
END_METHOD

END_FUNCTION_BLOCK

// ---- 01_Equipement_Library/Inverter/FB_INV_Base.TcPOU
FUNCTION_BLOCK FB_INV_Base
//////////////////
// PV INverter. Base FB. 
//////////////////

VAR_INPUT PERSISTENT
	// Parameters of the Object (instance/model specific) 
		ParamTempoComAlarm				: TIME := T#30S ; 			(* (s) Config : Tempo to detect LOC Alarm*)
		ParamTimeOutCurtail     		: TIME := T#45S ;			(* (s) Config : Tempo to curtail power at set value before Timeout warning*)
		{attribute 'OPC.UA.DA' := '1'} 
		ParamClockReadTime 				: TIME := TIME#2S;	  		(* (s) Read Modbus Frequency *)
		{attribute 'OPC.UA.DA' := '1'} 
		ParamClockWriteTime 			: TIME := TIME#500MS; 	  	(* (ms) Write Modbus Frequency *)
 		ParamTimeout					: TIME := T#5S ;		  	(* (s) Timeout for modbus reading *)
		ParamPn							: REAL ;      				(* (kW)   Nominal Capacity *)
		ParamQn							: REAL ;      				(* (kVAr) Nominal reactive power *)
		ParamPdc						: REAL;						(* (kWc) Power Crête use for power repartition *)
		ParamNumInv						: UINT;						(* (NA) Number of the Inverter*)

END_VAR

VAR_INPUT
		IN_SetptPlimit					: REAL;						// (kW) [P,H] Dynamic active Power limit setpoint (curtailing)  
		IN_SetptPlimit_Local			: REAL;						// (kW) [P,H] Dynamic active Power limit setpoint (curtailing)  
		IN_SetptQ						: REAL; 					// (kVar) Dynamic reactive power setpoints 	
		IN_CmdStart						: BOOL;						// (NA) [P,H] External Start Command
		IN_CmdStop 						: BOOL; 					// (NA) [P,H] External Stop Command 
		IN_CmdStop_Local				: BOOL; 					// (NA) [P,H] External Stop Command, only for this inverter
		IN_CmdStart_Local				: BOOL;						// (NA) [P,H] External Start Command, only for this inverter	
		                                                    		
		IN_CmdToggleRead				: BOOL ;            		
		IN_CmdToggleWrite				: BOOL ;            		
		IN_CmdReset_L					: BOOL ;					// (NA) External Reset Command
END_VAR

VAR
	// M_ALARMMNGMT VARIABLES //
		TON_ComAlarm				: TON ; 				// Tempo before deteting loss of communication. 
	    TON_ComWarning				: TON ; 				// Tempo before detecting loss of communication.                                                	
                                     		    	
		MesWarningCom				: BOOL ; 				// (NA) [P,H]  True if bad communication

		CalModbusWriteAlarm         : BOOL ; 				// (NA) Modbus Write Alarm synthesis


	// M_READ VARIABLES//
//	MesDataExd		      	: INV ; 				// (NA) [P,H,B] INV  Data Structure 


	// M_CURTAIL VARIABLES //
		FB_CheckCommand1		  	: FB_CheckCommand ; 	// (NA) Functionnal Block to check if Curtail limit Writing Successful
		FB_CheckSetPt		  		: FB_CheckSetPt ; 		// (NA) Functionnal Block to check if Q setpoint Writing Successful

		R_TRIG_Curtail				: R_TRIG ;

		CalCompareWarningCurtail	: BOOL ; 				// (NA) Curtail failed alarm						
		CalCompareWarningQSetpt		: BOOL ; 				// (NA) Curtail failed alarm						

		WriteCmdP 			 		: BOOL;					// Modbus Write Rising Edge 
		WriteCmdQ 			 		: BOOL;					// Modbus Write Rising Edge 
	

	// M_STARTSTOP//            	
		Trig_Cmd_Read				: R_TRIG; 
		Trig_Cmd_Write				: R_TRIG;  

		
		RS_Cmd_Read					: RS ; 	
		RS_Cmd_Write				: RS ; 	       	
		Trig_Local_Start			: R_Trig;
		Trig_Local_Stop				: R_Trig;
		Trig_Start					: R_Trig;
		Trig_Stop					: R_Trig;	         
		RS_StartStop				: RS ; 					// (NA) Bistable Function for Start and Stop 
		RS_StartStop_Local			: RS;					// (NA) Bistable Function for Start and Stop local                        	
		                       
	// M_STATEMANAGER//
		MesState					: BYTE ; 				// (NA) Cal [P,H,B] Bit 0: OFF , Bit 2 : Feeding Slave 	

	// M_CP VARIABLES //	
	
	//M_EXECUTE VARIABLES //
		TP1								: TP ; 				// (NA) Tempo to define Modbus Reading Frequency 
		TP2 							: TP ; 				// (NA) Tempo to define Modbus Writing Frequency
		
		ClockRead		AT %Q*				: BOOL;			// (NA) Modbus reading Clock
		ClockWrite 		AT %Q*				: BOOL;			// (NA) Modbus writing Clock 	
	
	//M_Init 
		bInit 							: BOOL := TRUE ; // Init variable	
		
		
		
		
		
END_VAR

METHOD M_AlarmManagement
//////////////////
// Manages IntelliGen Alarms
/////////////////

VAR 
	// Method local variables (reinitialized at each cycle) 

END_VAR
END_METHOD

METHOD M_CP
//////////////////
//  Emulator
/////////////////

VAR 
	// Method local variables (reinitialized at each cycle) 
	
END_VAR
END_METHOD

{attribute 'object_name' := 'M_Curtail'}
METHOD M_Curtail
//////////////////
// Write Curtail Command through modbus to PV inverters.  
//////////////////
VAR 
	// Method local variables (reinitialized at each cycle) 
	
	
END_VAR
IF IN_SetptPlimit	> IN_SetptPlimit_Local THEN
	IN_SetptPlimit := IN_SetptPlimit_Local;			// Local protection, can't take more than local setpoint
END_IF			
		

(*
// 	COMPARE CONSISTENCY	
	FB_CheckCommand1(
		T				:= ParamTimeOutCurtail ,
		bCmd			:= WriteCmdP, 
		bMes			:= MesDataExd.MesData.MesP < IN_SetptPlimit*1.05 , // 5% margin
		bImpulsion		:= TRUE , 
		bReset 			:= GVL_CFG.CmdClearFault_G, 
		bWarning 		=> CalCompareWarningCurtail); 
			
	FB_CheckSetPt(
			T					:= ParamTimeOutCurtail,
			Tolerance 			:= 5, 
			Range 				:= MesDataExd.MesData.ParamPn, 
			bTrigger 			:= WriteCmdQ , 
			bSetpt 				:= IN_SetptQlimit , 
			bMes 				:= MesDataExd.MesData.MesQ , 
			bReset				:= GVL_CFG.CmdClearFault_G  OR MesState <4 , 
			bWarning 			=> CalCompareWarningQSetpt);
			
			
			*)
END_METHOD

METHOD M_Execute
//////////////////
//  Method Calls 
/////////////////

VAR 
	// Method local variables (reinitialized at each cycle) 

END_VAR
// READING AND WRITING CLOCK //
	TP1(IN:=NOT TP1.Q , PT:= ParamClockReadTime);
	ClockRead 				:= TP1.Q;
	
	TP2(IN:=NOT TP2.Q , PT:= ParamClockWriteTime);
	ClockWrite 				:= TP2.Q;
	
// PERMANENT CONDITIONS //	
	M_CP() ; 
	
// METHODS CALLS//
	M_Read();

	M_StateManager() ; 
	M_StartStop() ; 
	M_Curtail();
	
	M_AlarmManagement();
END_METHOD

{attribute 'object_name' := 'M_Read'}
METHOD M_Read
//////////
// Read Method for SMA : Modbus reading
//////////
VAR
	// Method local variables (reinitialized at each cycle) 
	
END_VAR
END_METHOD

METHOD M_StartStop
//////////////////
// Start and Stop AMG
/////////////////
VAR 
	// Method local variables (reinitialized at each cycle) 

END_VAR
//IN_CmdStart := IN_CmdStart	AND NOT IN_CmdStop_Local; // Local Protection, can't switch on if i am switch off in local
END_METHOD

METHOD M_StateManager
//////////////////
// Detect which is the state of the inverter. IF loss of communication MesState =0 , the last inverter state is kept .  
/////////////////

VAR 
	// Method local variables (reinitialized at each cycle) 

	
END_VAR
END_METHOD

END_FUNCTION_BLOCK

// ---- 00_FunctionsBlocks/Common/AlarmManagement/FB_CheckCommand.TcPOU
FUNCTION_BLOCK FB_CheckCommand
////////////////// 
// Compare command with measure and raise warning if inconsistance. 
//////////////////	
VAR_INPUT
	T					: TIME ;			// Tempo to check if command has been executed	
	bCmd				: BOOL ; 			// Input command 
	bMes				: BOOL ; 			// Measure feedback 
	bReset				: BOOL := FALSE ; 	// Reset 
	bImpulsion			: BOOL ; 			// If True , the command is done on impulsion
	
END_VAR

VAR_OUTPUT
	bWarning 			: BOOL ; 		// Warning if inconsistancy . 
	bInProgress			: BOOL ; 		// Action in Progress
	
END_VAR

VAR

	// Inconsistency detection
	R_TRIG1				: R_TRIG ; 		// Detect command
	TOF1				: TOF ; 		// Creates a falling edge T time after command detcetion	
	F_TRIG				: F_TRIG ; 		// Detect Falling edge of TOF1	
	
	F_TRIG2				: F_TRIG ; 		// Detect falling edge of feedback measure
	TOF2				: TOF ; 		// Creates  a falling edge T time after Feedback measure ended detcetion
 
	TON					: TON ; 		// Tempo in case of bistable functuion

	// Reset management 	
	TOF_Reset			: TOF;			// Hold Reset command afetr reset to inhibate future warnings
	RS_Reset			: RS;			// Maintain reset command
	
END_VAR

IF bReset THEN
	bWarning 	:= FALSE ; 
END_IF

// Reset management 
TOF_Reset(IN:= bReset ,PT :=T);
RS_Reset(SET := bCmd,RESET1 := bReset) ; 


IF bImpulsion THEN 
	// Command is an impulsion
	R_TRIG1(CLK := bCmd) ; 
	TOF1(IN:=R_TRIG1.Q , PT:=T) ;
	F_TRIG(CLK:=TOF1.Q);		

	F_TRIG2(CLK := bMes) ;  
	TOF2(IN:=F_TRIG2.Q , PT:=T) ; 

ELSE
	// Command is a bistable function
	TON(IN:=bCmd , PT:= T);
END_IF

// Reset to False "InProgress" if Reset command or if command has been executed . 
bInProgress :=  ((TON.ET < TON.PT) AND (TON.ET>T#0S) OR (TOF1.ET < TOF1.PT) AND (TOF1.ET>T#0S)) AND NOT bMes AND RS_Reset.Q1  ; 

// Inconsistency detection
IF ((F_TRIG.Q AND NOT TOF2.Q AND NOT bMes) OR (TON.Q AND NOT bMes)) AND NOT TOF_Reset.Q  THEN
	bWarning := TRUE ; 
END_IF

END_FUNCTION_BLOCK

// ---- 00_FunctionsBlocks/Common/AlarmManagement/FB_CheckSetpt.TcPOU
FUNCTION_BLOCK FB_CheckSetpt
////////////////// 
// Compare SetPoint with measure and raise warning if inconsistance.
// The measure has to be within a range around the setpoint after a certain delay  . 
//////////////////	
VAR_INPUT
	T					: TIME ;		// Time to reacbh the range . 
	Tolerance			: INT := 5 ; 	// (%) Tolerance Window  
	Range 				: REAL ; 		// Maximal Range of the Setpoint
	bTrigger			: BOOL ; 		// Moment from which the setpoint is taken as reference
	bSetpt				: REAL ; 		// Input setpoint 
	bMes				: REAL ; 		// Measure feedback 
	bReset				: BOOL ; 		// Reset 
	
END_VAR

VAR_OUTPUT
	bWarning 			: BOOL ; 		// Warning if inconsistancy . 
	
END_VAR
VAR
	R_TRIG				: R_TRIG ; 		// Detect Trigger activation
	TOF					: TOF ; 		// Creates a falling edge T time after trigger activation
	F_TRIG				: F_TRIG ; 		// Detect end of timer. 
	
END_VAR

// Inconsistency detection

R_TRIG(CLK := bTrigger)  ;
TOF(IN := R_TRIG.Q , PT := T); 
F_TRIG(CLK := TOF.Q) ;


IF F_TRIG.Q AND ABS(bMes-bSetpt)>Tolerance/100*Range  THEN
	bWarning := TRUE ; 
END_IF

// Reset warning
IF bReset THEN
	bWarning := FALSE ; 
END_IF

END_FUNCTION_BLOCK

// ---- 00_FunctionsBlocks/Beckhoff/Communication/ModbusTCP/FB_ModbusRead.TcPOU
FUNCTION_BLOCK FB_ModbusRead
////////////////// 
// Read Modbus TCP/IP on Rising Edge of Trigger ClockRead. Returns alarm and stop modbus Read after three consecutive Modbus attempts that failed. 
//////////////////

VAR_INPUT
	
	// Modbus ReadRegs FB inputs
	pDestAddr 	: POINTER TO BYTE ; // Pointer to variable in which the read data have to be stored
	sIPAddr 	: STRING(15);		// Modbus server device IP adress
	tTimeout 	: TIME;				// Timeout
	nTcpPort 	: UINT;
	nQuantity 	: WORD;				// Quantity of words to be read
	nMBAddr 	: WORD ;			// Starting Register adress
	
	cbLength 	: UDINT;			// Length of variable to host the read data
	nUnitID 	: BYTE;				// Unit ID in case of serial connexion after modbus server. Usually equals to 1
	
	ClockRead	: BOOL; 			// Rising Edge Modbus Trigger
	Reset		: BOOL; 			// Reset Trigger to clean alarm and counter.
	
	ParamTimeRetry 			: TIME:=T#30S;				//Time to wait before a retry
	ParamNbAlms				: INT := 3;				// Parameter for the number of retries before the alarme
	ParamEnableRetryPause	: BOOL ; 
	
	
END_VAR

VAR_OUTPUT
	ErrorId			: UDINT;	// Error Id returned by FB ( see ADS error Code ) . 
	
	Busy			: BOOL ;	// FB busy to proceed command
	ModbusReadAlarm	: BOOL; 	// Alarm if three modbus attempt failed.
	OUT_NbRead		: UDINT;
END_VAR

VAR
	R_TRIG 				: R_TRIG; 			// Rising edge detection for the trigger.
	FB_MBReadRegs 		: FB_MBReadRegs; 	// Multiple registers reading
	
	Step				: INT; 				// Grafcet step
	AlarmCounter		: INT; 				// Alarm Counter. Incremennted if modbus errOR  Alarm if counter =3 , resetable.  

	TempoRetry      		: TP;

	bRetry          		: BOOL:= FALSE; 			// Boolean to denote the retries	
END_VAR

// ALARM MANAGEMENT //
TempoRetry(PT := ParamTimeRetry);
	IF AlarmCounter=ParamNbAlms THEN 
		ModbusReadAlarm 	:=TRUE;
		bRetry := SEL(ParamEnableRetryPause , FALSE ,  TRUE);		// False = disable retry 		
	ELSE
		ModbusReadAlarm := FALSE;
		ErrorId			:= 0;
		bRetry := FALSE;		// False = disable retry 	
	END_IF


// MODBUS SEQUENCE //
CASE Step OF 
	0:
		R_TRIG(CLK :=ClockRead);
		
		IF R_TRIG.Q THEN 
			Step :=1;
			Busy := TRUE;
			OUT_NbRead := 0;
		END_IF
	1:
	   FB_MBReadRegs(
	  			sIPAddr:= sIPAddr , 
				nTCPPort:= nTcpPort ,
				nUnitID:= nUnitID,
				nQuantity:= nQuantity,
				nMBAddr:= nMBAddr, 
				cbLength:= cbLength, 
				pDestAddr:= pDestAddr, 
				bExecute:= TRUE,
				tTimeout:= tTimeout,
				cbRead => OUT_NbRead
				);
				
		IF NOT FB_MBReadRegs.bBusy AND NOT FB_MBReadRegs.bError THEN
			FB_MBReadRegs(bExecute:= FALSE);
			AlarmCounter	:=0; // Reset counter after successful modbus read. 
			Step 			:=0;
			Busy := FALSE;
		ELSIF NOT FB_MBReadRegs.bBusy AND FB_MBReadRegs.bError AND NOT(bRetry) THEN
			FB_MBReadRegs(bExecute:= FALSE);
			AlarmCounter 	:= MIN(AlarmCounter+1,ParamNbAlms) ; 
			ErrorId			 :=FB_MBReadRegs.nErrId;
			Step 			:=0;
			Busy := FALSE;
			TempoRetry(In:= FALSE);
			bRetry := FALSE;
		ELSIF NOT FB_MBReadRegs.bBusy AND FB_MBReadRegs.bError AND bRetry THEN
			FB_MBReadRegs(bExecute:= FALSE);
			step := 2;
			Busy := FALSE;		
		END_IF	
	2: 
		TempoRetry(In:= TRUE);		// LEAVE SOME TIME BEFORE NEW ATTEMPT . 
		IF NOT(TempoRetry.Q) THEN
			TempoRetry(In:= FALSE);
			//AlarmCounter := 0;
			step := 0;
			
		END_IF
		
END_CASE

// RESET //
	IF Reset THEN 
			AlarmCounter 		:= 0 ; 
			ErrorId 			:= 0 ; 
			ModbusReadAlarm 	:=FALSE;
			Reset 				:= FALSE;
	END_IF

// BUSY //

END_FUNCTION_BLOCK

// ---- 00_FunctionsBlocks/Beckhoff/Communication/ModbusTCP/FB_ModbusWrite.TcPOU
FUNCTION_BLOCK FB_ModbusWrite
////////////////// 
// Write Modbus TCP/IP on Rising Edge of Trigger WriteCommAND  Returns alarm and stop modbus Read after three consecutive Modbus attempts that failed.
// Write two registers 
//////////////////
VAR_INPUT
	// Modbus ReadRegs FB inputs

	pSrcAddr			: POINTER TO BYTE ;
	sIPAddr 			: STRING(15);
	tTimeout 			: TIME;
	nTCPport			: UINT:= 502;		// TCP Port
	nMBAddr 			: WORD ;
	cbLength 			: UDINT ;
	nQuantity			: BYTE ;
	nUnitID 			: BYTE;
	WriteCmd 			: BOOL; 					// Rising Edge Trigger for sending modbus request
	
	Reset				: BOOL; 					// Reset Trigger to clean alarm and counter	
	
END_VAR


VAR_OUTPUT
	ErrorId				: UDINT; 			// Erreur ID returned by FB modbus. Updated every time on error occurs. 
	
	Completed			: BOOL ;			// Modbus Writing is completed 
	Busy				: BOOL ; 			// FB busy to proceed command
	ModbusWriteAlarm	: BOOL; 			// Alarm if three modbus attempt failed.
	
END_VAR
VAR
	R_TRIG 				: R_TRIG; 				// Rising edge detection for the trigger.
	FB_MBWriteRegs 		: FB_MBWriteRegs; 		// Multiple registers reading
	
	Step				: INT; 					// Grafcet step
	AlarmCounter		: INT; 					// Alarm Counter. Incremennted if modbus errOR  Alarm if counter =3 , resetable.  
END_VAR

Completed 				:= FALSE ;

// ALARM MANAGEMENT //
IF AlarmCounter=3 THEN
	ModbusWriteAlarm 	:=TRUE;
	
ELSE
	ModbusWriteAlarm 	:= FALSE;
	ErrorId				:= 0;
	
END_IF
	
// MODBUS SEQUENCE //
	CASE Step OF 
		0:
			R_TRIG(CLK :=WriteCmd);
			IF R_TRIG.Q THEN 
				Step :=1;
			END_IF
			
		1:
		   FB_MBWriteRegs(
					sIPAddr:= sIPAddr , 
					nTCPPort:= nTCPport ,
					nUnitID:= nUnitID,
					nQuantity:= nQuantity,
					nMBAddr:= nMBAddr, 
					cbLength:= cbLength, 
					pSrcAddr:= pSrcAddr, 
					bExecute:= TRUE,
					tTimeout:= tTimeout
					);
					
			IF NOT FB_MBWriteRegs.bBusy AND NOT FB_MBWriteRegs.bError THEN
				FB_MBWriteRegs(bExecute:= FALSE);
				AlarmCounter		:=0; // Reset counter after successful modbus read. 
				Step 				:=0;
				Completed 			:= TRUE ;
				
			ELSIF NOT FB_MBWriteRegs.bBusy AND FB_MBWriteRegs.bError THEN
				FB_MBWriteRegs(bExecute:= FALSE);
				AlarmCounter 		:=MIN(AlarmCounter+1,3) ; 
				ErrorId			 	:=FB_MBWriteRegs.nErrId;
				Step 				:=0;
				
			END_IF
			
	END_CASE

// RESET //	
	IF Reset THEN 
			AlarmCounter 	:= 0 ; 
			ErrorId 		:= 0 ; 
			Reset			:= FALSE;
	END_IF	
	
// BUSY //
	Busy 					:= FB_MBWriteRegs.bBusy ;

END_FUNCTION_BLOCK

// ---- 00_FunctionsBlocks/Common/AlarmManagement/FB_AlarmCodeManager.TcPOU
FUNCTION_BLOCK FB_AlarmCodeManager
////////////////// 
// Create Alarm Code from Alarms and Warnings conditions and summarize alarms
//////////////////	
VAR_INPUT
	bAlarm0				: BOOL:=FALSE; 			// Zero Alarm Condition (Optionnal only for subequipment)
	bAlarm1				: BOOL:=FALSE ; 		// First Alarm Condition  
	bAlarm2				: BOOL:=FALSE ; 		// Second Alarm Condition
	bAlarm3				: BOOL:=FALSE ; 		// Third Alarm Condition
	bAlarm4				: BOOL:=FALSE ; 		// Fourth Alarm Condition
	bAlarm5				: BOOL:=FALSE ; 		// Fifth Alarm Condition
	bAlarm6				: BOOL:=FALSE ; 		// First AlarmPermanent Condition
	bAlarm7				: BOOL:=FALSE ; 		// Second AlarmPermanent Condition
	bAlarm8				: BOOL:=FALSE ; 		// Third AlarmPermanent Condition
	bAlarm9				: BOOL:=FALSE ; 		// Fourth AlarmPermanent Condition 
	bAlarm10			: BOOL:=FALSE ; 		// Fourth AlarmPermanent Condition 
	bAlarm11			: BOOL:=FALSE ; 		// First AlarmPermanent Condition
	bAlarm12  			: BOOL:=FALSE ; 		// Second AlarmPermanent Condition
	bAlarm13			: BOOL:=FALSE ; 		// Third AlarmPermanent Condition
	bAlarm14			: BOOL:=FALSE ; 		// Fourth AlarmPermanent Condition 
	bAlarm15			: BOOL:=FALSE ; 		// Fourth AlarmPermanent Condition 

END_VAR

VAR_OUTPUT
	wAlarmCode		: WORD ; 		// 16 bit Alarm Code. 
END_VAR

VAR CONSTANT
	AlarmMask		: WORD := 2#1111111111111110 ;  // Alarm Mask 

	
END_VAR

// Reinitialize Alarm summary
wAlarmCode.0 := FALSE  ;

// Evaluate wAlarmCode
wAlarmCode.1 	:= bAlarm1 ;  
wAlarmCode.2 	:= bAlarm2 ;  
wAlarmCode.3 	:= bAlarm3 ;  
wAlarmCode.4 	:= bAlarm4 ;  
wAlarmCode.5 	:= bAlarm5 ;  
wAlarmCode.6 	:= bAlarm6 ; 
wAlarmCode.7 	:= bAlarm7 ; 
wAlarmCode.8 	:= bAlarm8 ;
wAlarmCode.9 	:= bAlarm9 ;
wAlarmCode.10 	:= bAlarm10 ; 
wAlarmCode.11 	:= bAlarm11 ; 
wAlarmCode.12 	:= bAlarm12 ; 
wAlarmCode.13 	:= bAlarm13 ; 
wAlarmCode.14 	:= bAlarm14 ; 
wAlarmCode.15 	:= bAlarm15 ; 
 
// Alarm Summarized
IF (AlarmMask AND wAlarmCode) >0 THEN
	wAlarmCode.0 := TRUE  ; 
END_IF

END_FUNCTION_BLOCK

// ---- 00_FunctionsBlocks/Common/DataProcessing/Split.TcPOU
PROGRAM Split
//Donne la position de la IN_Position-ième répétition du caractère recherché et renvoie la chaine de caractère suivante
VAR_INPUT
	IN_Delimiter 		: STRING;
	IN_TextToSearch		: T_MaxString;
END_VAR

VAR
	n					: UINT;	
	Position_Int		: UINT;
	LenOutSplit			: INT;
	TextToSearch_Int	: T_MaxString;
	OUT_Null			: ARRAY[1..100] OF T_Maxstring;
END_VAR

VAR_OUTPUT
	OUT_Split			: ARRAY[1..100] OF T_Maxstring;
	NbElements			: UINT;
END_VAR

OUT_Split := OUT_Null;
n:= 1;
TextToSearch_Int := IN_TextToSearch;
Position_Int := INT_TO_UINT( Find(STR1 := TextToSearch_Int, STR2 := IN_Delimiter));
LenOutSplit := 0;

WHILE Position_Int > 0 AND LenOutSplit < LEN(STR:= IN_TextToSearch) DO
	OUT_Split[n] := LEFT(STR := TextToSearch_Int, SIZE := UINT_TO_INT(Position_Int)-1);
	LenOutSplit := LenOutSplit + Len(STR := OUT_Split[n])+1;
	TextToSearch_Int := RIGHT(STR := TextToSearch_Int, SIZE := LEN(STR:= TextToSearch_Int)- LEN(STR:= OUT_Split[n])-1);
	Position_Int := INT_TO_UINT(FIND(STR1 := TextToSearch_Int, STR2 := IN_Delimiter));
	n := n + 1;
END_WHILE

NbElements := n-1;

END_PROGRAM

// ---- 00_FunctionsBlocks/Common/DataProcessing/SplitWord/FB_SplitRealToWords.TcPOU
FUNCTION_BLOCK FB_SplitRealToWords
////////////////// 
// Convert one REAL into  2 separate WORDS in Big Endian Encoding. 
//////////////////	
VAR_INPUT
	IN		: REAL ;				// Real input
	
END_VAR

VAR_OUTPUT
	OUT		: ARRAY[0..1]OF WORD;	// Word output array
	
END_VAR

OUT[1] := DWORD_TO_WORD(SHR(SHL(REAL_TO_DWORD(IN),16),16)) ; 	// Strong Word
OUT[0] := DWORD_TO_WORD(SHR(REAL_TO_DWORD(IN),16)); 			// Weak Word

END_FUNCTION_BLOCK

// ---- 00_FunctionsBlocks/Common/DataProcessing/MergeWord/FB_MergeWordsToDint.TcPOU
FUNCTION_BLOCK FB_MergeWordsToDint
////////////////// 
// Merge two words or one word into a DINT or UDINT with big endian coding. And finally Output a Real. 
//////////////////	

VAR_IN_OUT
	VAR_OUT 		: REAL ; 	
	
END_VAR

VAR_INPUT
	WORD_STRONG 	: WORD; 			// Strong Word. Word to consider if size equals 1.
	WORD_WEAK 		: WORD 	:= 0; 		// Weak Word. 
	
	SIZE 			: INT	:=1 ; 		// Nomber of words to considers. SIZE is equals to one (defaut) or two
	FIX 			: INT 	:=0 ; 		// Number of decimals (defaut 0)
	
	SIGNED 			: BOOL	:=FALSE; 	// Is the data signed or not (defaut) ? 
	SmaDevice 		: BOOL 	:= FALSE ; 	// True if device is SMA. 

END_VAR

VAR
	VAR_AUX 		: REAL ;			// Temporary variable before applying FIX
END_VAR

// Specific code to SMA 250000TL which provide weird data in case of no power on AC or DC Side
IF SmaDevice AND SIGNED AND (WORD_STRONG = 32768 OR WORD_STRONG = 65535)  THEN
		WORD_STRONG := 0 ;
		WORD_WEAK 	:= 0 ;
		
ELSIF SIGNED AND (WORD_STRONG = 32767 AND WORD_WEAK = 65535  )	THEN 	// Digiware 
		WORD_STRONG := 0 ;
		WORD_WEAK 	:= 0 ;

ELSIF WORD_STRONG=65535 AND WORD_WEAK = 65535 AND SIZE=2 AND NOT SIGNED THEN 
		WORD_STRONG := 0 ;
		WORD_WEAK 	:= 0 ;
		
ELSIF WORD_STRONG=65535 AND NOT SIGNED AND SIZE=1 THEN 
	WORD_STRONG := 0 ;

END_IF




IF SIGNED  THEN
	IF SIZE=2 THEN
		VAR_AUX := DINT_TO_REAL(DWORD_TO_DINT(SHL(WORD_TO_DWORD(WORD_STRONG),16) OR WORD_TO_DWORD(WORD_WEAK))) ; 
	ELSE
		VAR_AUX := INT_TO_REAL(WORD_TO_INT(WORD_STRONG)); 
	END_IF
ELSE
	IF SIZE=2 THEN
		VAR_AUX := DWORD_TO_REAL(SHL(WORD_TO_DWORD(WORD_STRONG),16) OR WORD_TO_DWORD(WORD_WEAK)) ;
	ELSE
		VAR_AUX := WORD_TO_REAL((WORD_STRONG));
	END_IF	
END_IF

VAR_OUT := VAR_AUX/(EXPT(10,FIX));

END_FUNCTION_BLOCK

// ---- 01_Equipement_Library/Inverter/FB_INV_Huawei_Sun2000KtlMo.TcPOU
FUNCTION_BLOCK FB_INV_Huawei_Sun2000KtlMo EXTENDS FB_INV_Base
// Huawei Sun2000 50KTL-M0. 
VAR_INPUT PERSISTENT
	// Parameters of the Object (instance specific)
	{attribute 'OPC.UA.DA' := '1'}  
	ParamIPAddress	   : STRING := '127.0.0.1'; 	(* (NA)Config: IP Adress of PV INverter*)
	{attribute 'OPC.UA.DA' := '1'} 	
	ParamTcpPort		: UINT := 502;				(* (NA)Modbus TCP port*)
	{attribute 'OPC.UA.DA' := '1'} 
	ParamUnitID 		: BYTE  := 1; 	  			(* (NA)   SMA Modbus Unit ID. *)
	ParamID_INV			: BYTE ; 		        	(* (NA) Config :Numerous of the ESS in the PP*)
	ParamID_PTR			: BYTE ; 		        	(* (NA) Config :Numerous of the ESS in the PP*)

END_VAR


VAR_INPUT 
			MesDataExd				AT %Q*	: INV_Huawei ; 
END_VAR

VAR_OUTPUT
	//Child objects

END_VAR

VAR
	//M_Acknowledge
		
	// M_ALARMMNGMT VARIABLES //
	MesAlarmCode1			: WORD ; 
	MesAlarmCode2			: WORD ; 
	
	// M_READ VARIABLES//
		Trig_Read					: R_TRIG;

		FB_ModbusRead_I2          	: FB_ModbusRead ; 									// (NA) FB for Modbus Reading
		FB_ModbusRead_I3          	: FB_ModbusRead ; 									// (NA) FB for Modbus Reading

		MesBlock_Temp 				: ARRAY[1..2] OF ARRAY [1..125] OF WORD ; 			// (NA) Temporary Block with multiple modbus reading (Caution : Double Word variables)

		AX_Busy						: ARRAY[1..2] OF BOOL;
		AX_Error					: ARRAY[1..2] OF BOOL;
		AX_ErrorID					: ARRAY[1..2] OF UDINT;



	// M_CP

		
	// M_STATEMANAGER//
	
	//M_EXECUTE VARIABLES //
		TP_READ						: LTP; 		//Tempo de cadencement FB Modbus
		RTrig						: R_Trig; 	//Front montant sur TP_READ.Q
		ReadBusy					: BOOL;		//FB Modbus en busy

	//M_CURTAIL 
	
		// M_CURTAIL VARIABLES //
	
		FB_ModbusWrite1 		  	: FB_ModbusWrite; 					// (NA) Functionnal Block for Writing Curtail limit through modbus
		FB_ModbusWrite2 		  	: FB_ModbusWrite; 					// (NA) Functionnal Block for Writing Curtail limit through modbus
	
		MesWriteBlock_Temp			: WORD;												// (NA) Temporary Block with multiple modbus writing	 
	
		MesModbusCurtailAlarm		: BOOL ;				   							// (NA) Modbus Write Curtail Alarm 
		MesModbusWriteCode          : UDINT ; 											// (NA) Modbus Write Alarm Code 			 
		
		WriteBlock_Temp1 				: WORD; 	// Temporary Block with multiple modbus writing	
		WriteBlock_Temp2 				: WORD; 	// Temporary Block with multiple modbus writing
		AX_Idc						: ARRAY[1..CstNbSB_INV_G] OF REAL;
		AX_TON_Idc_5percent			: ARRAY[1..CstNbSB_INV_G] OF TON;
		AX_TON_Idc_10percent		: ARRAY[1..CstNbSB_INV_G] OF TON;
		MesIdc_Median				: REAL;
		ParamTime5percent			: TIME := T#10M;
		ParamTime10percent			: TIME := T#10M;
	
	
END_VAR

METHOD M_AlarmManagement
//////////////////
// Manages IntelliGen Alarms
/////////////////

VAR 
	// Method local variables (reinitialized at each cycle) 
	FB_AlarmCodeManager : FB_AlarmCodeManager ; 

	KK					: BYTE;		// For Loop 
	

	ComAlarm: BOOL;
END_VAR
//COMMUNICATION//
// CALC INVERT STAT ERREUR //

ComAlarm :=AX_Error[1] OR AX_Error[2] ; 
TON_ComAlarm(IN:= ComAlarm , PT:= ParamTempoComAlarm, Q=>MesDataExd.MesData.MesAlarmCom) ;	

// ALARM CODE //
	FB_AlarmCodeManager(
		bAlarm1			:= MesDataExd.MesAlm1.0,		// High String Voltage #Equipment
		bAlarm2			:= MesDataExd.MesAlm1.1,		// DC Arc Fault #Equipment
		bAlarm3			:= MesDataExd.MesAlm1.2,		// String Reversed #Equipment
		bAlarm4			:= MesDataExd.MesAlm1.5, 	//    AFCI Self-test Fault    #Equipment 
		bAlarm5			:= MesDataExd.MesAlm1.6,	// Short circuit between phase to PE #Equipment
		bAlarm6			:= MesDataExd.MesAlm1.7,	 //Power Grid Failure #Equipment
		bAlarm7			:= MesDataExd.MesAlm1.8,     //Grid Undervoltage #Equipment
		bAlarm8			:= MesDataExd.MesAlm1.9,     //Grid Overvoltag #Equipment
		bAlarm9			:= MesDataExd.MesAlm1.10,    //Unbalanced Grid Voltage #Equipment
		bAlarm10		:= MesDataExd.MesAlm1.11,    //Grid Overfrequency #Equipment
		bAlarm11		:= MesDataExd.MesAlm1.12,    //Grid Underfrequency #Equipment
		bAlarm12		:= MesDataExd.MesAlm1.13,    //Grid Frequency Instability #Equipment
		bAlarm13		:= MesDataExd.MesAlm1.14,    //Output Overcurrent #Equipment
		bAlarm14		:= MesDataExd.MesAlm1.15, 	 //	Large DC of Output current	 #Equipment								
		bAlarm15		:= FALSE,//
		wAlarmCode		=> MesDataExd.MesData.MesAlarmCode);

// WARNING CODE //
	FB_AlarmCodeManager(
 		bAlarm1			:= MesDataExd.MesAlm2.0,//Abnormal Leakage Current #Equipment
		bAlarm2			:= MesDataExd.MesAlm2.1,//Abnormal Ground. #Equipment
		bAlarm3			:= MesDataExd.MesAlm2.2,//Low Insulation Res #Equipment
		bAlarm4			:= MesDataExd.MesAlm2.3,//High Temperature #Equipment
		bAlarm5			:= MesDataExd.MesAlm2.4,//Abnormal Equipment #Equipment
		bAlarm6			:= MesDataExd.MesAlm3.2,//High String Voltage to Ground #Equipment
		bAlarm7			:= MesDataExd.MesAlm2.5,//Upgrade Failed #Equipment
		bAlarm8			:= MesDataExd.MesAlm2.7,//Abnormal Monitor Unit #Equipment
		bAlarm9			:= MesDataExd.MesAlm3.1,//Built-in PID operation abnormal #Equipment
		bAlarm10		:= FALSE,//
		bAlarm11		:= FALSE,//
		bAlarm12		:= FALSE,//
		bAlarm13		:= FALSE,//
		bAlarm14		:= FALSE,//
		bAlarm15		:= MesDataExd.MesData.MesAlarmCom,//
		wAlarmCode		=> MesDataExd.MesData.MesWarningCode);	

// EVENT CODE //
	FB_AlarmCodeManager(
		bAlarm1			:= MesDataExd.MesAlm1.3, 			// PV String Backfeed #Equipment
		bAlarm2			:= MesDataExd.MesAlm1.4, 		// Abnormal String #Equipment
		bAlarm3			:= MesDataExd.MesAlm2.6,	// License Expired #Equipment
		bAlarm4			:= FALSE, 	
		bAlarm5			:= FALSE, 
		bAlarm6			:= FALSE, 
		bAlarm7			:= FALSE, 
		bAlarm8			:= FALSE, 
		bAlarm9			:= FALSE, 
		bAlarm10		:= FALSE, 
		bAlarm11		:= FALSE, 
		bAlarm12		:= FALSE, 
		bAlarm13		:= FALSE, 
		bAlarm14		:= FALSE, 
		bAlarm15		:= FALSE, 
		wAlarmCode		=> MesDataExd.MesData.MesEventCode);

(*

// ALARM CODE //
	FB_AlarmCodeManager(
		bAlarm0			:= , 	// standby
		bAlarm1			:= , 	// grid-connected
		bAlarm2			:= , 	// grid-connected normally
		bAlarm3			:= ,    // grid connection with derating due to power rationing
		bAlarm4			:= ,    // grid connection with derating due to internal causes of the solar inverter
		bAlarm5			:= ,    // normal stop
		bAlarm6			:= ,    // stop due to faults
		bAlarm7			:= ,    // stop due to power rationing
		bAlarm8			:= ,    // shutdown
		bAlarm9			:= ,    // spot check
		bAlarm10		:= ,    // 
		bAlarm11		:= ,    //
		bAlarm12		:= ,    //
		bAlarm13		:= ,    //
		bAlarm14		:= ,    //
		bAlarm15		:= ,	//
		wAlarmCode		=> MesDataExd.MesStateIndic);

// ALARM CODE //
	FB_AlarmCodeManager(
		bAlarm0			:= , 	// locking status (0: locked; 1: unlocked)
		bAlarm1			:= , 	// PV connection status (0: disconnected; 1: connected)
		bAlarm2			:= , 	// DSP data collection (0: no; 1: yes)
		bAlarm3			:= ,    // 
		bAlarm4			:= ,    // 
		bAlarm5			:= ,    // 
		bAlarm6			:= ,    // 
		bAlarm7			:= ,    // 
		bAlarm8			:= ,    // 
		bAlarm9			:= ,    // 
		bAlarm10		:= ,    // 
		bAlarm11		:= ,    //
		bAlarm12		:= ,    //
		bAlarm13		:= ,    //
		bAlarm14		:= ,    //
		bAlarm15		:= ,	//
		wAlarmCode		=> MesDataExd.MesOpeStatus);


*)
END_METHOD

METHOD M_CP
//////////////////
//  Emulator
/////////////////

VAR 
	// Method local variables (reinitialized at each cycle) 
	
END_VAR


SUPER^.M_CP() ; 




Trig_Cmd_Read(CLK:=IN_CmdToggleRead);
Trig_Cmd_Write(CLK:=IN_CmdToggleWrite);
	
IF Trig_Cmd_Read.Q THEN
	IN_CmdToggleRead := FALSE;
	MesDataExd.MesData.MesCP_Read := NOT MesDataExd.MesData.MesCP_Read;
END_IF


IF Trig_Cmd_Write.Q THEN
	IN_CmdToggleWrite := FALSE;
	MesDataExd.MesData.MesCP_Write := NOT MesDataExd.MesData.MesCP_Write;
END_IF
END_METHOD

{attribute 'object_name' := 'M_Curtail'}
METHOD M_Curtail
//////////////////
// Write Curtail Command through modbus to PV inverters.  
//////////////////
VAR 
	// Method local variables (reinitialized at each cycle) 
	SetptPlimit_Temp: WORD;
	SetptQlimit_Temp: WORD;	
	
	
	ClockWriteP: BOOL;
	ClockWriteQ: BOOL;
END_VAR


IF	MesDataExd.MesData.MesCP_Write THEN

// MODBUS VARIABLE FORMATING //
	IN_SetptPlimit := ParamPn;
	MesDataExd.MesData.OUT_SetptPLimit	:= MIN(100,MAX(0, (IN_SetptPlimit/ParamPn)*100)) ; //Between 0 and 100% Pmax
	MesDataExd.MesData.OUT_SetptQ	:= MIN(1 , MAX(-1 , IN_SetptQ/ParamPn)) ; //Between -1 and 1
	
	SetptPlimit_Temp := INT_TO_WORD(REAL_TO_INT(MesDataExd.MesData.OUT_SetptPLimit*10));
	SetptQlimit_Temp := INT_TO_WORD(REAL_TO_INT(MesDataExd.MesData.OUT_SetptQ*1000));
	
	IF SetptPlimit_Temp <> WriteBlock_Temp1 THEN
		ClockWriteP := TRUE;
		WriteBlock_Temp1 := SetptPlimit_Temp ; 
	END_IF
	IF SetptPlimit_Temp <> WriteBlock_Temp1 THEN
		ClockWriteQ := TRUE;
		WriteBlock_Temp2 := SetptQlimit_Temp ;  
	END_IF
	

	// MODBUS REQUEST //	
	// Modbus Blocks write
	
//	FB_ModbusWrite1(
//		pSrcAddr 			:= ADR(WriteBlock_Temp1), 
//		cbLength			:= SIZEOF(WriteBlock_Temp1),
//		nQuantity 			:= 1,
//		Reset				:=CmdClearFault_G, 
//		sIPAddr				:=ParamIPAddress ,
//		nTCPport			:=ParamTcpPort ,  
//		nUnitID				:=ParamUnitID , 
//		nMBAddr				:=40125 , 
//		tTimeout			:=ParamTimeout ,
//		WriteCmd			:=ClockWrite AND MesDataExd.MesData.MesCP_Write, 
//		ModbusWriteAlarm	=>MesModbusCurtailAlarm , 
//		ErrorId				=> MesModbusWriteCode); 
	
//	FB_ModbusWrite2(
//		pSrcAddr 			:= ADR(WriteBlock_Temp2), 
//		cbLength			:= SIZEOF(WriteBlock_Temp2),
//		nQuantity 			:= 1,
//		Reset				:=CmdClearFault_G, 
//		sIPAddr				:=ParamIPAddress ,
//		nTCPport			:=ParamTcpPort ,  
//		nUnitID				:=ParamUnitID , 
//		nMBAddr				:=40123 , 
//		tTimeout			:=ParamTimeout ,
//		WriteCmd			:=ClockWrite AND MesDataExd.MesData.MesCP_Write, 
//		ModbusWriteAlarm	=>MesModbusCurtailAlarm , 
//		ErrorId				=> MesModbusWriteCode);
		
		
	 

END_IF
END_METHOD

METHOD M_Init
VAR_INPUT
END_VAR

VAR

END_VAR
ParamPn := 60 ;

bInit := FALSE;
END_METHOD

{attribute 'object_name' := 'M_Read'}
METHOD M_Read
//////////
// Read Method for SMA : Modbus reading
//////////
VAR
	// Method local variables (reinitialized at each cycle) 
	KK					: BYTE;						 // Index to loop over modbus blocks. 	
	JJ					: BYTE;
	
	MW					: FB_MergeWordsToDint;
	
	
END_VAR
// Version table de com : Issu 02

IF MesDataExd.MesData.MesCP_Read THEN	

	//INITIALIZING MODBUS REQUESTS //

   //MODBUS REQUEST//
	FB_ModbusRead_I2(		
		nQuantity				:= 110, 
		nMBAddr					:= 32000, 
		cbLength				:= SIZEOF(MesBlock_Temp[1]) , 
		pDestAddr				:= ADR(MesBlock_Temp[1]) , 
		ClockRead				:= ClockRead AND MesDataExd.MesData.MesCP_Read,
		Reset					:= CmdClearFault_G ,
		sIPAddr					:= ParamIPAddress ,
		nUnitID					:= ParamUnitID, 
		tTimeout				:= ParamTimeout,
		nTcpPort 				:= ParamTcpPort, 
		ParamEnableRetryPause	:= FALSE,
		ModbusReadAlarm			=> AX_Error[1] , 
		ErrorId					=> AX_ErrorID[1]);

	
// MODBUS BLOCKS SEPARATION	
	MesdataExd.MesData.MesState_Inv:= MesBlock_Temp[1][1];


	//MesDataExd.MesData.MesState_Inv := MesBlock_Temp[1][1];
	MesDataExd.MesOpeStatus := MesBlock_Temp[1][3];
	MesDataExd.MesAlm1 := MesBlock_Temp[1][9];
	MesDataExd.MesAlm2 := MesBlock_Temp[1][10];
	MesDataExd.MesAlm3 := MesBlock_Temp[1][11];
	MesDataExd.MesDeviceStatus := MesBlock_Temp[1][90];
	
	FOR KK:=1  TO CstNbSB_INV_G DO 
		MW(WORD_STRONG := MesBlock_Temp[1][17+(KK-1)*2], FIX := 1, SIGNED := TRUE, VAR_OUT := MesdataExd.STR[KK].MesUdc	);
		MW(WORD_STRONG := MesBlock_Temp[1][17+(KK-1)*2+1], FIX := 2, SIGNED := TRUE, VAR_OUT := MesdataExd.STR[KK].MesIdc	);
	END_FOR
	
	MW(WORD_STRONG := MesBlock_Temp[1][65],WORD_WEAK := MesBlock_Temp[1][66], FIX := 3, Size := 2, SIGNED := TRUE, VAR_OUT := MesdataExd.Mesdata.MesPdc);
	MW(WORD_STRONG := MesBlock_Temp[1][67], FIX := 1, Size := 1, SIGNED := FALSE, VAR_OUT := MesdataExd.MesU12);
	MW(WORD_STRONG := MesBlock_Temp[1][68], FIX := 1, Size := 1, SIGNED := FALSE, VAR_OUT := MesdataExd.MesU23);
	MW(WORD_STRONG := MesBlock_Temp[1][69], FIX := 1, Size := 1, SIGNED := FALSE, VAR_OUT := MesdataExd.MesU31);
	MW(WORD_STRONG := MesBlock_Temp[1][70], FIX := 1, Size := 1, SIGNED := FALSE, VAR_OUT := MesdataExd.MesV1);
	MW(WORD_STRONG := MesBlock_Temp[1][71], FIX := 1, Size := 1, SIGNED := FALSE, VAR_OUT := MesdataExd.MesV2);
	MW(WORD_STRONG := MesBlock_Temp[1][72], FIX := 1, Size := 1, SIGNED := FALSE, VAR_OUT := MesdataExd.MesV3);
	MW(WORD_STRONG := MesBlock_Temp[1][73], WORD_WEAK := MesBlock_Temp[1][74], FIX := 3, Size := 2, SIGNED := TRUE, VAR_OUT := MesdataExd.MesI1);
	MW(WORD_STRONG := MesBlock_Temp[1][75], WORD_WEAK := MesBlock_Temp[1][76], FIX := 3, Size := 2, SIGNED := TRUE, VAR_OUT := MesdataExd.MesI2);
	MW(WORD_STRONG := MesBlock_Temp[1][77], WORD_WEAK := MesBlock_Temp[1][78], FIX := 3, Size := 2, SIGNED := TRUE, VAR_OUT := MesdataExd.MesI3);
	
	MW(WORD_STRONG := MesBlock_Temp[1][81], WORD_WEAK := MesBlock_Temp[1][82], FIX := 3, Size := 2, SIGNED := TRUE, VAR_OUT := MesdataExd.Mesdata.MesP);
	MW(WORD_STRONG := MesBlock_Temp[1][83], WORD_WEAK := MesBlock_Temp[1][84], FIX := 3, Size := 2, SIGNED := TRUE, VAR_OUT := MesdataExd.Mesdata.MesQ);
	MW(WORD_STRONG := MesBlock_Temp[1][85], FIX := 3, Size := 1, SIGNED := 1, VAR_OUT := MesDataExd.Mesdata.MesCosPhi);
	MW(WORD_STRONG := MesBlock_Temp[1][86], FIX := 2, Size := 1, SIGNED := 0, VAR_OUT := MesDataExd.Mesdata.MesFreq);
	MW(WORD_STRONG := MesBlock_Temp[1][88], FIX := 1, Size := 1, SIGNED := 0, VAR_OUT := MesDataExd.Mesdata.MesTemp);
	MW(WORD_STRONG := MesBlock_Temp[1][89], FIX := 0, Size := 1, SIGNED := 0, VAR_OUT := MesDataExd.Mesdata.MesInsuResistor);
	
	MW(WORD_STRONG := MesBlock_Temp[1][107], WORD_WEAK := MesBlock_Temp[1][108], FIX := 2, Size := 2, SIGNED := 0, VAR_OUT := MesdataExd.MesETot);
	MW(WORD_STRONG := MesBlock_Temp[1][109], WORD_WEAK := MesBlock_Temp[1][110], FIX := 2, Size := 2, SIGNED := 0, VAR_OUT := MesdataExd.MesEDay);

END_IF

// Properties update.
MesDataExd.MesData.MesI := (MesDataExd.MesI1 + MesDataExd.MesI2 + MesDataExd.MesI3)/3;
MesDataExd.MesData.MesV := (MesDataExd.MesV1 + MesDataExd.MesV2 + MesDataExd.MesV3)/3;
MesDataExd.MesData.MesU := (MesDataExd.MesU12 + MesDataExd.MesU23 + MesDataExd.MesU31)/3;
MesDataExd.MesData.MesS := SQRT(MesDataExd.MesData.MesP*MesDataExd.MesData.MesP + MesDataExd.MesData.MesQ*MesDataExd.MesData.MesQ);

MesDataExd.MesData.MesCurtl := MesDataExd.MesData.MesState=16#0201 OR MesDataExd.MesData.MesState =16#0202 ; 
MesDataExd.MesData.ParamPn := ParamPn ;


MesDataExd.MesData.MesIdc := 0;
MesDataExd.MesData.MesUdc := 0;

	FOR KK:=1  TO CstNbSB_INV_G DO 
		MesDataExd.MesData.MesIdc := MesDataExd.MesData.MesIdc + MesdataExd.STR[KK].MesIdc;
		MesDataExd.MesData.MesUdc := MesDataExd.MesData.MesUdc + MesdataExd.STR[KK].MesUdc/CstNbSB_INV_G;
	END_FOR
END_METHOD

METHOD M_StateManager
//////////////////
// Detect which is the state of the inverter. IF loss of communication MesState =0 , the last inverter state is kept .  
/////////////////

VAR 
	// Method local variables (reinitialized at each cycle) 

	
END_VAR

// 0 = Stopped, 1 = MPPT, 2 = Sleeping, 3 = Starting, 4 = Throttled, 5 = Shutting down, 6 = Fault, 7 = Standby

MesDataExd.Mesdata.MesState 			:= 0  ; 

IF     MesDataExd.MesData.MesState_Inv = 769 
	OR MesDataExd.MesData.MesState_Inv = 770
	OR MesDataExd.MesData.MesState_Inv = 771
	OR MesDataExd.MesData.MesState_Inv = 772
	OR MesDataExd.MesData.MesState_Inv = 773
	OR MesDataExd.MesData.MesState_Inv = 774 THEN // IF INVERTER IS STOPPED 309 = Operation && 455 = warning
	MesDataExd.Mesdata.MesState.0 := 1;		// Stop
ELSIF MesDataExd.MesData.MesState_Inv = 512 OR MesDataExd.MesData.MesState_Inv = 513 OR MesDataExd.MesData.MesState_Inv = 514 THEN
	MesDataExd.Mesdata.MesState.1 := 1;		// MPPT
ELSIF MesDataExd.MesData.MesState_Inv = 256 THEN
	MesDataExd.Mesdata.MesState.3 := 1;		// Starting
ELSIF MesDataExd.MesData.MesState_Inv = 0 OR MesDataExd.MesData.MesState_Inv = 1 OR MesDataExd.MesData.MesState_Inv = 2 OR MesDataExd.MesData.MesState_Inv = 3 OR MesDataExd.MesData.MesState_Inv = 16#A000  THEN
	MesDataExd.Mesdata.MesState.7 := 1;		// StandBy
ELSIF MesDataExd.MesData.MesState_Inv = 768  THEN
	MesDataExd.Mesdata.MesState.6 := 1;		// Fault
ELSIF MesDataExd.MesData.MesState_Inv = 16#201 OR MesDataExd.MesData.MesState_Inv = 16#202 THEN
	MesDataExd.Mesdata.MesState.4 := 1;		// Throlltled
ELSE 
	MesDataExd.Mesdata.MesState.1 := 1;
END_IF


SUPER^.M_StateManager() ;
END_METHOD

END_FUNCTION_BLOCK

// ---- 01_Equipement_Library/Inverter/FB_INV_JemaIFX6.TcPOU
FUNCTION_BLOCK FB_INV_JemaIFX6 EXTENDS FB_INV_Base


VAR_INPUT PERSISTENT
	// Parameters of the Object (instance specific) 
	ParamTcpPort				: UINT;			(*TCP Communication port*)
	ParamIpAddress				: STRING;       (*IP address*)
	ParamLVRT_Enabled			: BOOL;         (*Low Voltage Ride Through enabled*)
	ParamAntiIslanding_Enabled	: BOOL;         (*Anti Islanding enabled*)
	ParamRamp_Enabled			: BOOL;         (*Ramp enabled*)
	
	{attribute 'OPC.UA.DA' := '1'}		 
	ParamQoverP					: BOOL;         (*Q over P enabled*)
                      
END_VAR

VAR_INPUT
	MesOutputCbStatus_IO		: BOOL;      
	MesDataExd					: INV_Jema_IFX6;         		

END_VAR
VAR
	//M_Acknowledge
		
	// M_ALARMMNGMT VARIABLES //
	
	
	// M_READ VARIABLES//
		ModbusRead	          		: ARRAY[1..10] OF FB_ModbusRead; 	            // (NA) FB for Modbus Reading
		MesBlock_Temp 				: ARRAY[1..10] OF ARRAY [1..120] OF WORD ; 		// (NA) Temporary Block with multiple modbus reading (Caution : Double Word variables)
		AX_ModbusReadAlarm			: ARRAY[1..10] OF BOOL;
		AX_ModbusReadAlarmId		: ARRAY[1..10] OF UDINT;		
		
		ModbusWrite					: ARRAY[1..2] OF FB_ModbusWrite;
		AX_Cmd						: ARRAY[1..2] OF ARRAY[1..120] OF WORD;
		AX_ModbusWriteAlarm			: ARRAY[1..2] OF BOOL;
		AX_ModbusWriteAlarmId		: ARRAY[1..2] OF UDINT;
		
		
		
	
	// M_CURTAIL VARIABLES //
	

	// M_STARTSTOP//	                       	
		Trig_Cells					: R_TRIG;
		Trig_CmdP					: R_TRIG;
		Trig_CmdQ					: R_TRIG;
		Trig_CmdPF					: R_TRIG;
		Trig_CmdPvF					: R_TRIG;
		Trig_CmdQvU					: R_TRIG;
		
		
		CmdCells_IO					: BOOL;		// Input for the control of the cells (toggle)
		CmdP_IO						: BOOL;		// Input for the control of the P mode (toggle)
		CmdQ_IO						: BOOL;		// Input for the control of the Q mode (toggle)
		CmdPF_IO					: BOOL;		// Input for the control of the PF mode (toggle)
		CmdStart_IO					: BOOL;
		CmdStop_IO					: BOOL; 
		CmdPvF_IO 					: BOOL; 	// Input for the control of the PvF function(toggle)
		CmdQvU_IO 					: BOOL; 	// Input for the control of the PvF function(toggle)
	
	// M_CP

	
	//M_EXECUTE VARIABLES //
		TP_READ						: LTP;  //Tempo de cadencement FB Modbus
		RTrig						: R_Trig; //Front montant sur TP_READ.Q
		ReadBusy					: BOOL;	//FB Modbus en busy
		
END_VAR

METHOD M_Acknowledge
VAR
		//Each cycle
	Temp_Alarm	:BOOL:=False;	
END_VAR
END_METHOD

METHOD M_AlarmManagement
//////////////////
// Manages IntelliGen Alarms
/////////////////

VAR 
	// Method local variables (reinitialized at each cycle) 
	FB_AlarmCodeManager : FB_AlarmCodeManager ; 
	KK				: BYTE;		// For Loop 
	bComError		: BOOL := TRUE;
	bComWarning 	: BOOL;

	MesComWarning: BOOL;
END_VAR
MesDataExd.mesData.MesAlarmCom := ModbusRead[1].ModbusReadAlarm AND ModbusRead[2].ModbusReadAlarm AND ModbusRead[3].ModbusReadAlarm AND ModbusRead[4].ModbusReadAlarm AND ModbusRead[5].ModbusReadAlarm AND ModbusRead[6].ModbusReadAlarm AND ModbusRead[7].ModbusReadAlarm AND ModbusRead[8].ModbusReadAlarm AND ModbusRead[9].ModbusReadAlarm AND ModbusRead[10].ModbusReadAlarm AND ModbusWrite[1].ModbusWriteAlarm;
MesComWarning := ModbusRead[1].ModbusReadAlarm OR ModbusRead[2].ModbusReadAlarm OR ModbusRead[3].ModbusReadAlarm OR ModbusRead[4].ModbusReadAlarm OR ModbusRead[5].ModbusReadAlarm OR ModbusRead[6].ModbusReadAlarm OR ModbusRead[7].ModbusReadAlarm OR ModbusRead[8].ModbusReadAlarm OR ModbusRead[9].ModbusReadAlarm OR ModbusRead[10].ModbusReadAlarm OR ModbusWrite[1].ModbusWriteAlarm;



// ALARM CODE //
	FB_AlarmCodeManager(
		bAlarm1			:= MesDataExd.mesData.MesAlarmCom,		// Communication alarm (all frames failed)
		bAlarm2			:= MesComWarning,	// Communication Warning (at least on frame failed)
		bAlarm3			:= ( MesDataExd.AX_PowerCol[1].MesRegAlarm0 > 0 OR MesDataExd.AX_PowerCol[2].MesRegAlarm0 > 0 OR MesDataExd.AX_PowerCol[3].MesRegAlarm0 > 0 ),		// INV : Alarm0 > 0 on one module
		bAlarm4			:= MesDataExd.AX_PowerCol[1].MesRegAlarm1 > 0  OR MesDataExd.AX_PowerCol[2].MesRegAlarm1 > 0  OR MesDataExd.AX_PowerCol[3].MesRegAlarm1 > 0  ,		// INV : Alarm1 > 0 on one module
		bAlarm5			:= MesDataExd.AX_PowerCol[1].MesRegAlarm2 > 0 OR MesDataExd.AX_PowerCol[2].MesRegAlarm2 > 0 OR MesDataExd.AX_PowerCol[3].MesRegAlarm2 > 0,			// INV : Alarm2 > 0 on one module
		bAlarm6			:= (MesDataExd.AX_PowerCol[1].MesRegAlarm3 > 0 AND MesDataExd.AX_PowerCol[1].MesRegAlarm3 <> 160) OR ( MesDataExd.AX_PowerCol[2].MesRegAlarm3 > 0 AND MesDataExd.AX_PowerCol[2].MesRegAlarm3 <> 160) OR (MesDataExd.AX_PowerCol[3].MesRegAlarm3 > 0 AND MesDataExd.AX_PowerCol[3].MesRegAlarm3 <> 160),		// INV : Alarm3 > 0 on one module
		bAlarm7			:= MesDataExd.AX_PowerCol[1].MesRegAlarm4 > 0 OR MesDataExd.AX_PowerCol[2].MesRegAlarm4 > 0 OR MesDataExd.AX_PowerCol[3].MesRegAlarm4 > 0,			// INV : Alarm4 > 0 on one module
		bAlarm8			:= MesDataExd.MesPLC_IN1 > 0,																											// INV : Input1 > 0 
		bAlarm9			:= MesDataExd.MesPLC_IN2 > 0,																											// INV : Input2 > 0 
		bAlarm10		:= MesOutputCbStatus_IO,					// Output CB Status IO
		bAlarm11		:= FALSE,
		bAlarm12		:= FALSE,
		bAlarm13		:= FALSE,
		bAlarm14		:= FALSE,
		bAlarm15		:= False,
		wAlarmCode		=> MesDataExd.mesData.MesAlarmCode);
END_METHOD

METHOD M_CP
//////////////////
//  Emulator
/////////////////

VAR 
	// Method local variables (reinitialized at each cycle) 
	
END_VAR


SUPER^.M_CP() ; 




Trig_Cmd_Read(CLK:=IN_CmdToggleRead);
Trig_Cmd_Write(CLK:=IN_CmdToggleWrite);
	
IF Trig_Cmd_Read.Q THEN
	IN_CmdToggleRead := FALSE;
	MesDataExd.MesData.MesCP_Read := NOT MesDataExd.MesData.MesCP_Read;
END_IF


IF Trig_Cmd_Write.Q THEN
	IN_CmdToggleWrite := FALSE;
	MesDataExd.MesData.MesCP_Write := NOT MesDataExd.MesData.MesCP_Write;
END_IF
END_METHOD

{attribute 'object_name' := 'M_Curtail'}
METHOD M_Curtail
//////////////////
// Write Curtail Command through modbus to PV inverters.  
//////////////////
VAR 
	// Method local variables (reinitialized at each cycle) 


	
	AX_ADDR				: ARRAY[1..2] OF UINT := [1800, 623];
	AX_QTY				: ARRAY[1..2] OF BYTE := [11, 	1];
	AX_UnitId			: ARRAY[1..2] OF BYTE := [1, 	1];

	KK: INT;
	Word_To_Write : WORD;
END_VAR
SUPER^.M_Curtail() ; 

MesDataExd.OUT_SetptP := MAX(0, MIN(ParamPn, IN_SetptPlimit));
MesDataExd.OUT_SetptQ := MAX(-ParamPn, MIN(ParamPn, IN_SetptQ));

MesDataExd.OUT_SetptQMax       := SQRT(ABS((ParamPn*ParamPn) - (MesDataExd.MesData.MesP*MesDataExd.MesData.MesP)));
MesDataExd.OUT_SetptQMin       := -MesDataExd.OUT_SetptQMax;

IF MesDataExd.OUT_SetptQ < MesDataExd.OUT_SetptQMin   THEN
	MesDataExd.OUT_SetptQ      := MesDataExd.OUT_SetptQMin;
END_IF

IF MesDataExd.OUT_SetptQ > MesDataExd.OUT_SetptQMax THEN
	MesDataExd.OUT_SetptQ      :=  MesDataExd.OUT_SetptQMax;
END_IF

// MODBUS VARIABLE FORMATING //
	AX_Cmd[1][1] := BOOL_TO_WORD(MesDataExd.OUT_CmdP);
	AX_Cmd[1][2] := BOOL_TO_WORD(MesDataExd.OUT_CmdQ);
	AX_Cmd[1][3] := REAL_TO_WORD(MesDataExd.OUT_SetptP);
	AX_Cmd[1][4] := REAL_TO_WORD(-MesDataExd.OUT_SetptQ);
	AX_Cmd[1][5] := BOOL_TO_WORD(MesDataExd.OUT_CmdPF);
	AX_Cmd[1][6] := REAL_TO_WORD(MesDataExd.OUT_SetptPF*1000);
	AX_Cmd[1][7] := BOOL_TO_WORD(NOT MesDataExd.OUT_CmdStart);
	AX_Cmd[1][8] := 1;
	AX_Cmd[1][9] := BOOL_TO_WORD(NOT MesDataExd.OUT_CmdCells);	
	AX_Cmd[1][10] := MesDataExd.OUT_CmdControl;	
	AX_Cmd[1][11] := BOOL_TO_WORD(MesDataExd.OUT_CmdHeartBeat);
	
Modbuswrite[1]
(
	pSrcAddr 			:= ADR(AX_Cmd[1]),
	sIPAddr 			:= ParamIPAddress,
	tTimeout 			:= ParamTimeout,
	nTCPport 			:= ParamTcpPort,
	nMBAddr 			:= AX_ADDR[1],
	cbLength 			:= SIZEOF(AX_CMd[1]),
	nQuantity 			:= AX_QTY[1],
	nUnitID 			:= AX_UnitId[1],
	WriteCmd 			:= ClockWrite and MesDataExd.Mesdata.MesCP_Write,
	ModbusWriteAlarm 	=> AX_ModbusWriteAlarm[1],
	ErrorId 			=> AX_ModbusWriteAlarmId[1]
);
END_METHOD

METHOD M_Execute
//////////////////
//  Method Calls 
/////////////////

VAR 
	// Method local variables (reinitialized at each cycle) 

END_VAR
IF NOT bInit THEN
	M_Init();
END_IF

SUPER^.M_Execute() ;
END_METHOD

METHOD M_Init
VAR_INPUT
END_VAR

VAR
	bCompleted : BOOL := FALSE;
END_VAR
IN_SetptPlimit_Local := ParamPn;

Trig_Cmd_Read(CLK:=TRUE);
Trig_Cmd_Write(CLK:=TRUE);

bInit := true;
END_METHOD

{attribute 'object_name' := 'M_Read'}
METHOD M_Read
//////////
// Read Method for SMA : Modbus reading
//////////
VAR
	// Method local variables (reinitialized at each cycle) 
	//MW					: FB_MergeWordsToFloat;
	//MW_1				: FB_WordsToDint64BE;
	

	MW					: FB_MergeWordsToDint;
	AX_QTY_MB			: ARRAY[1..10] OF WORD := [82,	68, 	68, 	68, 	1,		6, 		28,		2,		1,		25];
	AX_ADR_MB			: ARRAY[1..10] OF WORD := [5,	100, 	200, 	300, 	623, 	1005,	1110,	1298,	1500, 	2020];
	AX_UnitID			: ARRAY[1..10] OF BYTE := [1, 	1,		1,		1, 		1,		1,		1,		1,		1,		1];
	TimeInterm			: REAL;
	U_dc_Temp			: REAL:=0;
	Nbr_CbDC			: REAL:=0;
	PosInterm: REAL;
	KK : UINT;
END_VAR

IF MesDataExd.MesData.MesCP_Read THEN
	FOR KK := 1 TO 10 DO 
		ModbusRead[KK]
		(
			nTCPPort		:= ParamTcpPort,
			ClockRead		:= ClockRead, 
			Reset			:= CmdClearFault_G ,
			sIPAddr			:=ParamIPAddress ,
			nUnitID			:= AX_UnitID[KK], 
			tTimeout		:= ParamTimeout,
			nQuantity		:= AX_QTY_MB[KK] , 
			nMBAddr			:= AX_ADR_MB[KK] , 
			cbLength		:= SIZEOF(MesBlock_Temp[KK]) , 
			pDestAddr		:= ADR(MesBlock_Temp[KK]) , 
			ModbusReadAlarm	=>AX_ModbusReadAlarm[KK] , 
			ErrorId			=> AX_ModbusReadAlarmId[KK]
		);
	END_FOR
		
    
	// BLOCK1 1
		MW(WORD_STRONG :=  MesBlock_Temp[1][1],											SIZE := 1, 	FIX := 1, 	SIGNED := 0, 	VAR_OUT	:= MesDataExd.Mesdata.mesPdc);
		MW(WORD_STRONG :=  MesBlock_Temp[1][77],WORD_STRONG :=  MesBlock_Temp[1][78],	SIZE := 2, 	FIX := 2, 	SIGNED := 0, 	VAR_OUT	:= MesDataExd.MesEacTot);
		MW(WORD_STRONG :=  MesBlock_Temp[1][79],WORD_STRONG :=  MesBlock_Temp[1][80],	SIZE := 2, 	FIX := 1, 	SIGNED := 0, 	VAR_OUT	:= MesDataExd.MesEacDay);

	// BLOCK 2, 3 et 4
	
		MesDataExd.MesPowerColConnected_ALO := FALSE;
		MesDataExd.MesNbPowerCol_Connected := 0 ; 
	
	
		FOR KK := 2 TO 4 DO
			MW(WORD_STRONG :=  MesBlock_Temp[KK][ 1],											SIZE := 1, 	FIX := 1, 	SIGNED := 1, 	VAR_OUT	:= MesDataExd.AX_PowerCol[KK-1].MesData.MesUdc);
			MW(WORD_STRONG :=  MesBlock_Temp[KK][ 2],											SIZE := 1, 	FIX := 1, 	SIGNED := 1, 	VAR_OUT	:= MesDataExd.AX_PowerCol[KK-1].MesData.MesIdc);
			MW(WORD_STRONG :=  MesBlock_Temp[KK][ 3],											SIZE := 1, 	FIX := 1, 	SIGNED := 0, 	VAR_OUT	:= MesDataExd.AX_PowerCol[KK-1].MesData.MesV1);
			MW(WORD_STRONG :=  MesBlock_Temp[KK][ 4],											SIZE := 1, 	FIX := 1, 	SIGNED := 0, 	VAR_OUT	:= MesDataExd.AX_PowerCol[KK-1].MesData.MesV2);
			MW(WORD_STRONG :=  MesBlock_Temp[KK][ 5],											SIZE := 1, 	FIX := 1, 	SIGNED := 0, 	VAR_OUT	:= MesDataExd.AX_PowerCol[KK-1].MesData.MesV3);
			MW(WORD_STRONG :=  MesBlock_Temp[KK][ 6],											SIZE := 1, 	FIX := 1, 	SIGNED := 1, 	VAR_OUT	:= MesDataExd.AX_PowerCol[KK-1].MesData.MesI1);
			MW(WORD_STRONG :=  MesBlock_Temp[KK][ 7],											SIZE := 1, 	FIX := 1, 	SIGNED := 1, 	VAR_OUT	:= MesDataExd.AX_PowerCol[KK-1].MesData.MesI2 );
			MW(WORD_STRONG :=  MesBlock_Temp[KK][ 8],											SIZE := 1, 	FIX := 1, 	SIGNED := 1, 	VAR_OUT	:= MesDataExd.AX_PowerCol[KK-1].MesData.MesI3);
			MW(WORD_STRONG :=  MesBlock_Temp[KK][ 9],											SIZE := 1, 	FIX := 1, 	SIGNED := 1, 	VAR_OUT	:= MesDataExd.AX_PowerCol[KK-1].MesData.MesPdc);
			MW(WORD_STRONG :=  MesBlock_Temp[KK][10],											SIZE := 1, 	FIX := 1, 	SIGNED := 1, 	VAR_OUT	:= MesDataExd.AX_PowerCol[KK-1].MesData.MesP);
			MW(WORD_STRONG :=  MesBlock_Temp[KK][11],											SIZE := 1, 	FIX := 1, 	SIGNED := 1, 	VAR_OUT	:= MesDataExd.AX_PowerCol[KK-1].MesData.MesQ);
			MW(WORD_STRONG :=  MesBlock_Temp[KK][12],											SIZE := 1, 	FIX := 3, 	SIGNED := 1, 	VAR_OUT	:= MesDataExd.AX_PowerCol[KK-1].MesData.MesCosPhi);
			MW(WORD_STRONG :=  MesBlock_Temp[KK][13],											SIZE := 1, 	FIX := 2, 	SIGNED := 0, 	VAR_OUT	:= MesDataExd.AX_PowerCol[KK-1].MesData.MesFreq);
			MW(WORD_STRONG :=  MesBlock_Temp[KK][15],											SIZE := 1, 	FIX := 1, 	SIGNED := 0, 	VAR_OUT	:= MesDataExd.AX_PowerCol[KK-1].MesTempControl);
			MesDataExd.AX_PowerCol[KK-1].MesIn_State 	:= MesBlock_Temp[KK][16];
			MesDataExd.AX_PowerCol[KK-1].MesOut_State 	:=  MesBlock_Temp[KK][17];
			MW(WORD_STRONG :=  MesBlock_Temp[KK][18],											SIZE := 1, 	FIX := 1, 	SIGNED := 0, 	VAR_OUT	:= MesDataExd.AX_PowerCol[KK-1].MesTempPowerUnit);
			MW(WORD_STRONG :=  MesBlock_Temp[KK][20],											SIZE := 1, 	FIX := 1, 	SIGNED := 0, 	VAR_OUT	:= MesDataExd.AX_PowerCol[KK-1].MesTempCabinet);
			
			//Update des Alarmes modules
				MesDataExd.AX_PowerCol[KK-1].MesRegAlarm0		:=		MesBlock_Temp[KK][24];
				MesDataExd.AX_PowerCol[KK-1].MesJemaAlarms.MesI1_Alm			   := MesDataExd.AX_PowerCol[KK-1].MesRegAlarm0.0;
				MesDataExd.AX_PowerCol[KK-1].MesJemaAlarms.MesI2_Alm			   := MesDataExd.AX_PowerCol[KK-1].MesRegAlarm0.1;
				MesDataExd.AX_PowerCol[KK-1].MesJemaAlarms.MesI3_Alm			   := MesDataExd.AX_PowerCol[KK-1].MesRegAlarm0.2;
				MesDataExd.AX_PowerCol[KK-1].MesJemaAlarms.MesVdc_High_Alm		   := MesDataExd.AX_PowerCol[KK-1].MesRegAlarm0.3;
				MesDataExd.AX_PowerCol[KK-1].MesJemaAlarms.MesVdc_Low_Alm		   := MesDataExd.AX_PowerCol[KK-1].MesRegAlarm0.4;
				MesDataExd.AX_PowerCol[KK-1].MesJemaAlarms.MesU12_High_Alm		   := MesDataExd.AX_PowerCol[KK-1].MesRegAlarm0.6;
				MesDataExd.AX_PowerCol[KK-1].MesJemaAlarms.MesU12_Low_Alm		   := MesDataExd.AX_PowerCol[KK-1].MesRegAlarm0.7;
				MesDataExd.AX_PowerCol[KK-1].MesJemaAlarms.MesU23_High_Alm		   := MesDataExd.AX_PowerCol[KK-1].MesRegAlarm0.8;
				MesDataExd.AX_PowerCol[KK-1].MesJemaAlarms.MesU23_Low_Alm		   := MesDataExd.AX_PowerCol[KK-1].MesRegAlarm0.9;
				MesDataExd.AX_PowerCol[KK-1].MesJemaAlarms.MesU31_High_Alm		   := MesDataExd.AX_PowerCol[KK-1].MesRegAlarm0.10;
				MesDataExd.AX_PowerCol[KK-1].MesJemaAlarms.MesU31_Low_Alm		   := MesDataExd.AX_PowerCol[KK-1].MesRegAlarm0.11;
				MesDataExd.AX_PowerCol[KK-1].MesJemaAlarms.MesVdc_Neg		   := MesDataExd.AX_PowerCol[KK-1].MesRegAlarm0.14;
				MesDataExd.AX_PowerCol[KK-1].MesJemaAlarms.MesIdc_Neg		   := MesDataExd.AX_PowerCol[KK-1].MesRegAlarm0.15;
				
				MesDataExd.AX_PowerCol[KK-1].MesRegAlarm1   	:=      MesBlock_Temp[KK][25];
				MesDataExd.AX_PowerCol[KK-1].MesJemaAlarms.MesU1223_Unbalance	:= MesDataExd.AX_PowerCol[KK-1].MesRegAlarm1.0;
				MesDataExd.AX_PowerCol[KK-1].MesJemaAlarms.MesU2331_Unbalance	:= MesDataExd.AX_PowerCol[KK-1].MesRegAlarm1.1;
				MesDataExd.AX_PowerCol[KK-1].MesJemaAlarms.MesU3112_Unbalance	:= MesDataExd.AX_PowerCol[KK-1].MesRegAlarm1.2;
				MesDataExd.AX_PowerCol[KK-1].MesJemaAlarms.MesInvertedPhase	  	:= MesDataExd.AX_PowerCol[KK-1].MesRegAlarm1.3;
				MesDataExd.AX_PowerCol[KK-1].MesJemaAlarms.MesI12_Unbalance	  	:= MesDataExd.AX_PowerCol[KK-1].MesRegAlarm1.4;
				MesDataExd.AX_PowerCol[KK-1].MesJemaAlarms.MesI23_Unbalance	  	:= MesDataExd.AX_PowerCol[KK-1].MesRegAlarm1.5;
				MesDataExd.AX_PowerCol[KK-1].MesJemaAlarms.MesI31_Unbalance	  	:= MesDataExd.AX_PowerCol[KK-1].MesRegAlarm1.6;
				MesDataExd.AX_PowerCol[KK-1].MesJemaAlarms.MesF_High			:= MesDataExd.AX_PowerCol[KK-1].MesRegAlarm1.8;
				MesDataExd.AX_PowerCol[KK-1].MesJemaAlarms.MesF_Low			    := MesDataExd.AX_PowerCol[KK-1].MesRegAlarm1.9;
				MesDataExd.AX_PowerCol[KK-1].MesJemaAlarms.MesPcbOverTemp		:= MesDataExd.AX_PowerCol[KK-1].MesRegAlarm1.12;

				
				MesDataExd.AX_PowerCol[KK-1].MesRegAlarm2   	:=      MesBlock_Temp[KK][26];
				MesDataExd.AX_PowerCol[KK-1].MesJemaAlarms.MesGridCbOpened			:= MesDataExd.AX_PowerCol[KK-1].MesRegAlarm2.4;
				MesDataExd.AX_PowerCol[KK-1].MesJemaAlarms.MesGridCbTrip	  		:= MesDataExd.AX_PowerCol[KK-1].MesRegAlarm2.5;
				MesDataExd.AX_PowerCol[KK-1].MesJemaAlarms.MesGridContactFail 		:= MesDataExd.AX_PowerCol[KK-1].MesRegAlarm2.8;
				MesDataExd.AX_PowerCol[KK-1].MesJemaAlarms.MesDoorOpened			:= MesDataExd.AX_PowerCol[KK-1].MesRegAlarm2.9;
				MesDataExd.AX_PowerCol[KK-1].MesJemaAlarms.MesAuxCbOpened 			:= MesDataExd.AX_PowerCol[KK-1].MesRegAlarm2.13;
				MesDataExd.AX_PowerCol[KK-1].MesJemaAlarms.MesOverVoltHyst			:= MesDataExd.AX_PowerCol[KK-1].MesRegAlarm2.14;
				MesDataExd.AX_PowerCol[KK-1].MesJemaAlarms.MesIdcMax				:= MesDataExd.AX_PowerCol[KK-1].MesRegAlarm2.15;
	
				
				MesDataExd.AX_PowerCol[KK-1].MesRegAlarm3   	:=      MesBlock_Temp[KK][27];
				
				MesDataExd.AX_PowerCol[KK-1].MesJemaAlarms.MesSKIIP1				 	:= MesDataExd.AX_PowerCol[KK-1].MesRegAlarm3.0;
				MesDataExd.AX_PowerCol[KK-1].MesJemaAlarms.MesSKIIP2				 	:= MesDataExd.AX_PowerCol[KK-1].MesRegAlarm3.1;
				MesDataExd.AX_PowerCol[KK-1].MesJemaAlarms.MesSKIIP3				 	:= MesDataExd.AX_PowerCol[KK-1].MesRegAlarm3.2;
				MesDataExd.AX_PowerCol[KK-1].MesJemaAlarms.MesSKIIP_OT				 	:= MesDataExd.AX_PowerCol[KK-1].MesRegAlarm3.3;
				MesDataExd.AX_PowerCol[KK-1].MesJemaAlarms.MesHardwareOverCurrent		:= MesDataExd.AX_PowerCol[KK-1].MesRegAlarm3.4;
				MesDataExd.AX_PowerCol[KK-1].MesJemaAlarms.MesCoilOverTemp				:= MesDataExd.AX_PowerCol[KK-1].MesRegAlarm3.11;
				MesDataExd.AX_PowerCol[KK-1].MesJemaAlarms.MesAlrmGrp1_Curr		  		:= MesDataExd.AX_PowerCol[KK-1].MesRegAlarm3.13;
				MesDataExd.AX_PowerCol[KK-1].MesJemaAlarms.MesAlrmGrp2_Curr		  		:= MesDataExd.AX_PowerCol[KK-1].MesRegAlarm3.14;
				MesDataExd.AX_PowerCol[KK-1].MesJemaAlarms.MesShortCircuit_DC			:= MesDataExd.AX_PowerCol[KK-1].MesRegAlarm3.15;
				
				MesDataExd.AX_PowerCol[KK-1].MesRegAlarm4   		:=      MesBlock_Temp[KK][28];
					// States
				MesDataExd.AX_PowerCol[KK-1].MesData.MesAcSwitchClosed 		:= MesDataExd.AX_PowerCol[KK-1].MesIn_State.1 ;	// AC contactor status
				MesDataExd.AX_PowerCol[KK-1].MesDeratingWord 		:= MesBlock_Temp[KK][62] ;
				MesDataExd.MesPowerColConnected_ALO 				:= MesDataExd.MesPowerColConnected_ALO OR MesDataExd.AX_PowerCol[KK-1].MesData.MesAcSwitchClosed ;
				
				MesDataExd.MesNbPowerCol_Connected			:= MesDataExd.MesNbPowerCol_Connected + SEL(MesDataExd.AX_PowerCol[KK-1].MesData.MesAcSwitchClosed , 0,1) ; 
			
				
			//Inversion signe de la puissance reactive.
			MesDataExd.AX_PowerCol[KK-1].MesData.MesQ	:= - MesDataExd.AX_PowerCol[KK-1].MesData.MesQ;
		END_FOR                                                                                                                                                                		

	
	// BLOCK 5
		MesDataExd.MesGFDI := MesBlock_Temp[5][1];
	// BLOCK 6
		MW(WORD_STRONG :=  MesBlock_Temp[6][1],											SIZE := 1, 	FIX := 1, 	SIGNED := 0, 	VAR_OUT	:= MesDataExd.MesI1);
		MW(WORD_STRONG :=  MesBlock_Temp[6][2],											SIZE := 1, 	FIX := 1, 	SIGNED := 0, 	VAR_OUT	:= MesDataExd.MesI2);
		MW(WORD_STRONG :=  MesBlock_Temp[6][3],											SIZE := 1, 	FIX := 1, 	SIGNED := 0, 	VAR_OUT	:= MesDataExd.MesI3);
		MW(WORD_STRONG :=  MesBlock_Temp[6][5],											SIZE := 1, 	FIX := 1, 	SIGNED := 1, 	VAR_OUT	:= MesDataExd.MesData.MesP);
		MW(WORD_STRONG :=  MesBlock_Temp[6][6],											SIZE := 1, 	FIX := 1, 	SIGNED := 1, 	VAR_OUT	:= MesDataExd.MesData.MesQ);
		MesDataExd.MesData.MesQ	:= -MesDataExd.MesData.MesQ;
		
	// BLOCK 7
		FOR KK := 1 TO 24 DO
			MW(WORD_STRONG :=  MesBlock_Temp[7][KK],									SIZE := 1, 	FIX := 2, 	SIGNED := 0, 	VAR_OUT	:= MesDataExd.AX_STR[KK].MesIdc);
		END_FOR
		
		MW(WORD_STRONG :=  MesBlock_Temp[7][25],									SIZE := 1, 	FIX := 0, 	SIGNED := 0, 	VAR_OUT	:= MesDataExd.MesTmpPlant);
		MW(WORD_STRONG :=  MesBlock_Temp[7][26],									SIZE := 1, 	FIX := 1, 	SIGNED := 0, 	VAR_OUT	:= MesDataExd.MesVdc1);
		MW(WORD_STRONG :=  MesBlock_Temp[7][27],									SIZE := 1, 	FIX := 1, 	SIGNED := 0, 	VAR_OUT	:= MesDataExd.MesVdc2);
		MW(WORD_STRONG :=  MesBlock_Temp[7][28],									SIZE := 1, 	FIX := 1, 	SIGNED := 0, 	VAR_OUT	:= MesDataExd.MesVdc3);
	
	// BLOCK 8 
		MesDataExd.MesPLC_IN1 				:= MesBlock_Temp[8][1];
		MesDataExd.MesPLC_IN2 				:= MesBlock_Temp[8][2];
		
	// BLOCK 9
		MesDataExd.MesData.MesInsuResistor := WORD_TO_REAL(MesBlock_Temp[9][1]	);
	
	// BLOCK 10	
		MW(WORD_STRONG :=  MesBlock_Temp[10][1 ],											SIZE := 1, 	FIX := 1, 	SIGNED := 0, 	VAR_OUT	:= MesDataExd.MesTmpExt1);
		MW(WORD_STRONG :=  MesBlock_Temp[10][2 ],											SIZE := 1, 	FIX := 1, 	SIGNED := 0, 	VAR_OUT	:= MesDataExd.MesTmpExt2);
		MW(WORD_STRONG :=  MesBlock_Temp[10][3 ],											SIZE := 1, 	FIX := 1, 	SIGNED := 0, 	VAR_OUT	:= MesDataExd.MesTmp);
		MW(WORD_STRONG :=  MesBlock_Temp[10][4 ],											SIZE := 1, 	FIX := 1, 	SIGNED := 0, 	VAR_OUT	:= MesDataExd.MesTmpPlc);
		MW(WORD_STRONG :=  MesBlock_Temp[10][5 ],											SIZE := 1, 	FIX := 1, 	SIGNED := 0, 	VAR_OUT	:= MesDataExd.MesHygroPlc);
		
		IF MesDataExd.MesData.MesP <> 0 THEN
			MesDataExd.MesPowerColConnected_ALO := TRUE;
		END_IF


//MesDataUpdate 
		MesDataExd.MesData.ParamPn 	:= ParamPn;
		MesDataExd.MesData.MesS := SQRT(MesDataExd.MesData.MesP*MesDataExd.MesData.MesP + MesDataExd.MesData.MesQ*MesDataExd.MesData.MesQ);

		MesDataExd.MesData.MesUdc := (MesDataExd.MesVdc1 + MesDataExd.MesVdc2) / 2 ; 


	MesDataExd.MesData.MesIdc := 0 ; 
	FOR KK:=1 TO 3 DO 
		MesDataExd.MesData.MesIdc:=MesDataExd.MesData.MesIdc  + MesDataExd.AX_PowerCol[KK].MesData.MesIdc ; 
	END_FOR	
END_IF
END_METHOD

METHOD M_StartStop
VAR_INPUT
END_VAR
VAR
	KK : UINT;
	AX_ADR_MB			: ARRAY[1..2] OF WORD := [11600, 21600];
	AX_QTY_MB			: ARRAY[1..2] OF BYTE := [2, 2];
	MotStart			: WORD := 1467;
	MotStop				: WORD := 1749;
	
END_VAR
SUPER^.M_StartStop() ; 




IF IN_CmdStart_Local THEN 
	IN_CmdStart_Local := FALSE;
	MesDataExd.OUT_CmdStart := TRUE;
END_IF
IF IN_CmdStop_Local THEN
	IN_CmdStop_Local := FALSE;
	MesDataExd.OUT_CmdStart := FALSE;
	
END_IF


IF CmdCells_IO THEN
	CmdCells_IO := FALSE;
	MesDataExd.OUT_CmdCells := NOT MesDataExd.OUT_CmdCells;
END_IF

IF CmdP_IO THEN
	CmdP_IO := FALSE;
	MesDataExd.OUT_CmdP := NOT MesDataExd.OUT_CmdP;
END_IF

IF CmdQ_IO THEN
	CmdQ_IO := FALSE;
	MesDataExd.OUT_CmdQ := NOT MesDataExd.OUT_CmdQ;
	MesDataExd.OUT_CmdPF := NOT MesDataExd.OUT_CmdPF;
END_IF

IF CmdPF_IO THEN
	CmdPF_IO := FALSE;
	MesDataExd.OUT_CmdQ := NOT MesDataExd.OUT_CmdQ;
	MesDataExd.OUT_CmdPF := NOT MesDataExd.OUT_CmdPF;
END_IF



MesDataExd.OUT_CmdHeartBeat := CalLocalTimeStruct.wSecond MOD 2 > 0;

MesDataExd.OUT_CmdControl.0 := ParamLVRT_Enabled ;
MesDataExd.OUT_CmdControl.1 := MesDataExd.OUT_CmdQvU;
MesDataExd.OUT_CmdControl.2 := MesDataExd.OUT_CmdPvF;
MesDataExd.OUT_CmdControl.3 := ParamAntiIslanding_Enabled;
MesDataExd.OUT_CmdControl.4 := MesDataExd.OUT_CmdQ;
MesDataExd.OUT_CmdControl.5 := MesDataExd.OUT_CmdPF;
MesDataExd.OUT_CmdControl.7 := ParamQoverP;
MesDataExd.OUT_CmdControl.9 := ParamRamp_Enabled;
END_METHOD

METHOD M_StateManager
//////////////////
// Detect which is the state of the inverter. IF loss of communication MesState =0 , the last inverter state is kept .  
/////////////////

VAR 
	// Method local variables (reinitialized at each cycle) 

	
END_VAR
//O=Stopped, 1 = MPPT, 2 = Sleeping, 3 = Starting, 4 = Throttled, 5 = Shutting down, 6 = Fault, 7 = Standby

SUPER^.M_StateManager() ; 

MesDataExd.MesData.MesState := 0;


IF NOT MesDataExd.MesPowerColConnected_ALO THEN
	MesDataExd.MesData.MesState.6 := TRUE;  // Fault 
ELSIF MesDataExd.MesPowerColConnected_ALO THEN
	IF MesDataExd.MesData.MesP > 0.01  THEN
		MesDataExd.MesData.MesState.1 := TRUE; // Ongrid 
	ELSE
		MesDataExd.MesData.MesState.7 := TRUE; // Standby 
	END_IF
	

END_IF
END_METHOD

END_FUNCTION_BLOCK

// ---- 01_Equipement_Library/Inverter/FB_INV_Power_One.TcPOU
FUNCTION_BLOCK FB_INV_Power_One EXTENDS FB_INV_Base
//////////////////
// Power One ( ABB) inverters ) 
// PT1: 
// PT2: 18 BJ
// PT3:	
// PT4: 18 BJ
//////////////////
VAR_INPUT PERSISTENT
	// Parameters of the Object (instance specific) 

	(* ajouter parametres ID pour les fct modbus *)
	ParamUnitID 				: BYTE  := 1; 			  (* (NA)   SMA Modbus Unit ID. *)
	ParamFunctionReadModbus		: BYTE := 4 ; (* (NA)   Modbus Function. *)
	Master_slave_Calculation 	: BOOL; //Gestion de la soustraction des modules
	WriteTest					: UINT := 0;
	
END_VAR


VAR_INPUT
	
	IN_SetptTanPhi				: REAL ; // (p.u) Setpt Tanphi 
	MesDataExd					: INV_ClusterPowerOne;
END_VAR


VAR_OUTPUT
	//Child objects

	OUT_CmdSetpt420_IO				: INT;

END_VAR

VAR
	// M_ALARMMNGMT VARIABLES //
	
	// M_READ VARIABLES//

		FB_ModbusRTU	          	: FB_ModbusRTU; 	            // (NA) FB for Modbus Reading

		RTrigI						: R_TRIG;
		InputStructRead 			: Struct_InputRTU ; 
		InputStructRead_Null		: Struct_InputRTU ; 
		bReadCompleted 				: BOOL;

		InverterNumber				: BYTE;
		Steps						: INT:=1;
		MesBlock_Temp 				: ARRAY[1..18] OF ARRAY [0..66] OF WORD ; 			// (NA) Temporary Block with multiple modbus reading (Caution : Double Word variables)
		MesBlock_Temp_Anemo			: ARRAY[0..128] OF WORD;
		AX_bRead 					: ARRAY[0..18] OF BOOL; 
		CalAllCompleted				: BOOL; 
		CalAllBugged				: BOOL; 
		TON_AllBugged				: TON;
		TRIG_AllBugged				: R_TRIG;
		
		ReadError					: BOOL; //FB Modbus en error

		AX_Start_Adresse			: ARRAY [1..18] OF WORD :=[228,328,428,528,628,728,828,928,1028,1128,1228,1328,1428,1528,1628,1728,1828,1928];  // First Module 228, 7module 628
		DecalageInvModule			: INT;
		MesTempPSlave				: ARRAY [1..9] OF ARRAY [1..4] OF REAL;
		MesTempPMaster				: ARRAY [1..9] OF ARRAY [1..4] OF REAL;
		MesTempPos					: ARRAY [1..9] OF INT;
		Nb_DataBlockModules			: WORD:=65;

	// M_INIT //
		OutFBCompleteted 	        : BOOL;
	
	// M_STARTSTOP//
	// M_CP
	// M_STATEMANAGER//
	
	//M_EXECUTE VARIABLES //
		TP_READ						: LTP;  //Tempo de cadencement FB Modbus
		RTrig						: R_Trig; //Front montant sur TP_READ.Q
		ReadBusy					: BOOL;	//FB Modbus en busy
	//EMULATOR VARIABLES //




		
END_VAR

METHOD M_Acknowledge
VAR
		//Each cycle
	Temp_Alarm	:BOOL:=False;	
END_VAR
END_METHOD

METHOD M_AlarmManagement
//////////////////
// Manages IntelliGen Alarms
/////////////////

VAR 
	// Method local variables (reinitialized at each cycle) 
	FB_AlarmCodeManager : FB_AlarmCodeManager ; 
	InvWarning		: ARRAY [1..3] OF BOOL;
	InvAlarm		: ARRAY [1..3] OF BOOL;
	KK				: BYTE;		// For Loop 
	

END_VAR
//COMMUNICATION//
// CALC INVERT STAT ERREUR //
	//INV 1
		InvWarning[1]	:= MesDataExd.AX_INV[1].AX_PowerCol[1].MesAlarmID > 0 OR MesDataExd.AX_INV[1].AX_PowerCol[2].MesAlarmID > 0 OR MesDataExd.AX_INV[1].AX_PowerCol[3].MesAlarmID > 0 
							OR MesDataExd.AX_INV[1].AX_PowerCol[4].MesAlarmID > 0 OR MesDataExd.AX_INV[1].AX_PowerCol[5].MesAlarmID > 0 OR MesDataExd.AX_INV[1].AX_PowerCol[6].MesAlarmID > 0;
		InvAlarm[1]		:= MesDataExd.AX_INV[1].AX_PowerCol[1].MesAlarmID > 0 AND MesDataExd.AX_INV[1].AX_PowerCol[2].MesAlarmID > 0 AND MesDataExd.AX_INV[1].AX_PowerCol[3].MesAlarmID > 0 
							AND MesDataExd.AX_INV[1].AX_PowerCol[4].MesAlarmID > 0 AND MesDataExd.AX_INV[1].AX_PowerCol[5].MesAlarmID > 0 AND MesDataExd.AX_INV[1].AX_PowerCol[6].MesAlarmID > 0;
	//INV 2
		InvWarning[2]	:= MesDataExd.AX_INV[2].AX_PowerCol[1].MesAlarmID > 0 OR MesDataExd.AX_INV[2].AX_PowerCol[2].MesAlarmID > 0 OR MesDataExd.AX_INV[2].AX_PowerCol[3].MesAlarmID > 0 
							OR MesDataExd.AX_INV[2].AX_PowerCol[4].MesAlarmID > 0 OR MesDataExd.AX_INV[2].AX_PowerCol[5].MesAlarmID > 0 OR MesDataExd.AX_INV[2].AX_PowerCol[6].MesAlarmID > 0;
		InvAlarm[2]		:= MesDataExd.AX_INV[2].AX_PowerCol[1].MesAlarmID > 0 AND MesDataExd.AX_INV[2].AX_PowerCol[2].MesAlarmID > 0 AND MesDataExd.AX_INV[2].AX_PowerCol[3].MesAlarmID > 0 
							AND MesDataExd.AX_INV[2].AX_PowerCol[4].MesAlarmID > 0 AND MesDataExd.AX_INV[2].AX_PowerCol[5].MesAlarmID > 0 AND MesDataExd.AX_INV[2].AX_PowerCol[6].MesAlarmID > 0;	
	//INV 3
		InvWarning[3]	:= MesDataExd.AX_INV[3].AX_PowerCol[1].MesAlarmID > 0 OR MesDataExd.AX_INV[3].AX_PowerCol[2].MesAlarmID > 0 OR MesDataExd.AX_INV[3].AX_PowerCol[3].MesAlarmID > 0 
							OR MesDataExd.AX_INV[3].AX_PowerCol[4].MesAlarmID > 0 OR MesDataExd.AX_INV[3].AX_PowerCol[5].MesAlarmID > 0 OR MesDataExd.AX_INV[3].AX_PowerCol[6].MesAlarmID > 0;
		InvAlarm[3]		:= MesDataExd.AX_INV[3].AX_PowerCol[1].MesAlarmID > 0 AND MesDataExd.AX_INV[3].AX_PowerCol[2].MesAlarmID > 0 AND MesDataExd.AX_INV[3].AX_PowerCol[3].MesAlarmID > 0 
							AND MesDataExd.AX_INV[3].AX_PowerCol[4].MesAlarmID > 0 AND MesDataExd.AX_INV[3].AX_PowerCol[5].MesAlarmID > 0 AND MesDataExd.AX_INV[3].AX_PowerCol[6].MesAlarmID > 0;
	
						

	//Warning
	MesWarningCom 	:= ReadError ;  

